METHOD PRIVATE FlagOpenEntity : BOOL
VAR_INPUT
	Identifier : STRING(255);	
END_VAR
VAR_IN_OUT
	Header : CuHeader;
END_VAR
Header.Operator := _operatorInfo.UserName;
Header.OperationsStarted := Context.RealTimeClock.NowLocal();
THIS^.ProcessDataManager.Data.EntityHeader.Results.Result := TcoInspectors.eOverallResult.InProgress;
THIS^.ProcessDataManager.Data._EntityId := Identifier;
THIS^.ProcessDataManager.Data.EntityHeader.OpenOn := THIS^.CuId;
THIS^.ProcessDataManager.Data.EntityHeader.WasReset := FALSE;
END_METHOD

METHOD PRIVATE FlagThrowAwayEntity : BOOL
VAR_IN_OUT	
	CuHeader : CuHeader; 
END_VAR
IF(THIS^.ProcessDataManager.Data.EntityHeader.OpenOn <> eStations.NONE) THEN
	THIS^.ProcessDataManager.Data.EntityHeader.LastStation := THIS^.CuId;
	THIS^.ProcessDataManager.Data.EntityHeader.NextStation := CuHeader.NextOnFailed;
	THIS^.ProcessDataManager.Data.EntityHeader.Results.Result := TcoInspectors.eOverallResult.Failed;
	THIS^.ProcessDataManager.Data.EntityHeader.WasReset := TRUE;
END_IF;
END_METHOD

(*~
	<docu>
		<summary>
			Controls `ground` mode of `CU00x`.
		</summary>
	</docu>
~*)
METHOD Ground : BOOL
VAR_INPUT
END_VAR
(*
	Enable condition to start `groundTask`.
	Modify according your needs.
	[! 
	THIS IS NOT SAFETY CONDITION. THE SAFETY OF PRESONNEL AND EQUIPMENT MUST BE ENSURED BY ADDITIONAL MEANS 
	TO COMPLY WITH REGULATIONS
	]
*)

GroundTask.Task.Enabled :=  THIS^.Technology.AllowGround(inCuId:=CuId)  OR GroundTask.Task.Busy ;

(*
	Invokes `groundTask` from technology object.
*)


IF(Technology.GroundAllTask.Execute()) THEN GroundTask.Restore();GroundTask.Task.Invoke(); END_IF;


IF GroundTask.GroundDone AND GroundTask.Task.Execute() THEN GroundTask.Restore();GroundTask.Task.Invoke();END_IF;
END_METHOD

PROPERTY ABSTRACT GroundTask : REFERENCE TO CUBaseGround
GET
END_GET
END_PROPERTY

PROPERTY FINAL GroupInspection : REFERENCE TO TcoInspectionGroup
GET
GroupInspection REF= _groupInspection;
END_GET
END_PROPERTY

(*~
	<docu>
		<summary>
			Code to be called cylically when `CU00x` idle; no other mode is active.
		</summary>
	</docu>
~*)
METHOD Idle : BOOL
END_METHOD

METHOD InternalCloseEntity : BOOL
VAR_INPUT
	inCarrier : UINT;
	refStorage : REFERENCE TO InternalStorage;
END_VAR
VAR_IN_OUT
	inoHeader : CuHeader; 
END_VAR
VAR_INST
	_internalData : REFERENCE TO InternalStorage;	
END_VAR
THIS^.FlagCloseEntity(inoHeader);
_internalData REF= refStorage;
InternalCloseEntity := _internalData.SaveByCarrier(inCarrier, THIS^.ProcessDataManager.Data);
END_METHOD

METHOD InternalCreateNewEntity : BOOL
VAR_INPUT
	inCarrier : UINT;
	refStorage : REFERENCE TO InternalStorage;
END_VAR
VAR_IN_OUT
	inoHeader : CuHeader; 
END_VAR
VAR_INST
	_internalData : REFERENCE TO InternalStorage;	
END_VAR
THIS^.FlagCreateNewEntity(UINT_TO_STRING(inCarrier), inoHeader);
THIS^.ProcessDataManager.Data.EntityHeader.Carrier := UINT_TO_STRING(inCarrier);
_internalData REF= refStorage;
InternalCreateNewEntity := _internalData.SaveByCarrier(inCarrier, THIS^.ProcessDataManager.Data);
END_METHOD

METHOD InternalFinishEntity : BOOL
VAR_INPUT
	inCarrier : UINT;
	refStorage : REFERENCE TO InternalStorage;
END_VAR
VAR_IN_OUT
	inoHeader : CuHeader; 
END_VAR
VAR_INST
	_internalData : REFERENCE TO InternalStorage;	
END_VAR
THIS^.FlagFinishEntity(inoHeader);

_internalData REF= refStorage;
InternalFinishEntity := _internalData.SaveByCarrier(inCarrier, THIS^.ProcessDataManager.Data);
END_METHOD

METHOD InternalOpenEntity : BOOL
VAR_INPUT
	inCarrier : UINT;
	refStorage : REFERENCE TO InternalStorage;
END_VAR
VAR_IN_OUT
	inoHeader : CuHeader; 
END_VAR
VAR_INST
	_internalData : REFERENCE TO InternalStorage;	
END_VAR
_internalData REF= refStorage;
InternalOpenEntity := _internalData.GetByCarrier(inCarrier, THIS^.ProcessDataManager.Data);
THIS^.FlagOpenEntity(UINT_TO_STRING(inCarrier), inoHeader);
END_METHOD

METHOD InternalRetrieveEntity : BOOL
VAR_INPUT
	inCarrier : UINT;
	refStorage : REFERENCE TO InternalStorage;
END_VAR
VAR_INST
	_internalData : REFERENCE TO InternalStorage;	
END_VAR
_internalData REF= refStorage;
InternalRetrieveEntity := _internalData.GetByCarrier(inCarrier, THIS^.ProcessDataManager.Data);
END_METHOD

METHOD InternalThrowAwayEntity : BOOL
VAR_INPUT
	inCarrier : UINT;
	refStorage : REFERENCE TO InternalStorage;
END_VAR
VAR_IN_OUT
	inoHeader : CuHeader; 
END_VAR
VAR_INST
	_internalData : REFERENCE TO InternalStorage;	
END_VAR
THIS^.FlagThrowAwayEntity(inoHeader);
_internalData REF= refStorage;
InternalThrowAwayEntity := _internalData.SaveByCarrier(inCarrier, THIS^.ProcessDataManager.Data);
END_METHOD

(*~
	<docu>
		<summary>
			Controls `manual` mode of `CU00x`.
		</summary>
	</docu>
~*)
METHOD Manual : BOOL
VAR_INPUT
END_VAR
(*
	Enable condition to start `automatTask`.
	Modify according your needs.
	[! 
	THIS IS NOT SAFETY CONDITION. THE SAFETY OF PRESONNEL AND EQUIPMENT MUST BE ENSURED BY ADDITIONAL MEANS 
	TO COMPLY WITH REGULATIONS
	]
*)

ManualTask.Task.Enabled :=  THIS^.Technology.AllowManual(inCuId:=CuId)  OR ManualTask.Task.Busy;
END_METHOD

PROPERTY ABSTRACT ManualTask : REFERENCE TO TcoTaskedService
GET
END_GET
END_PROPERTY

PROPERTY FINAL ProcessDataManager : REFERENCE TO ProcessDataManager
GET
ProcessDataManager REF= _processData;
END_GET
END_PROPERTY

PROPERTY  ReadEntityTask : TcoCore.ITcoTaskStatus
GET
ReadEntityTask := _processData._readTask;
END_GET
END_PROPERTY

METHOD ReadyForOperations : BOOL
VAR_INPUT
END_VAR
ReadyForOperations := _readyForOperations;
END_METHOD

PROPERTY ABSTRACT RecoverTask : REFERENCE TO CUBaseRecover
GET
END_GET
END_PROPERTY

PROPERTY RecurringFails : REFERENCE TO CuBaseRecurringFailures
GET
RecurringFails REF= _recurringFails;
END_GET
END_PROPERTY

METHOD ResetReadyForOperations : BOOL
_readyForOperations := false;
END_METHOD

METHOD  RunOperations : BOOL
VAR_INPUT
	refGlobalTrigger:REFERENCE TO BOOL;
END_VAR
VAR
	_trrigger:REFERENCE TO BOOL;
END_VAR
_trrigger REF=refGlobalTrigger;
RunOperations := _trrigger;
END_METHOD

METHOD  SetReadyForOperations : BOOL
VAR_INPUT
END_VAR
_readyForOperations := TRUE;
END_METHOD

PROPERTY ABSTRACT StatusInfo : REFERENCE TO CUBaseStatusInfo
GET
END_GET
END_PROPERTY

PROPERTY ABSTRACT SuspendTask : REFERENCE TO CUBaseSuspend
GET
END_GET
END_PROPERTY

PROPERTY Technology : REFERENCE TO Technology
GET
VAR
    _technology : POINTER TO Technology;
END_VAR
IF __QUERYPOINTER(Parent, _technology) THEN // Check if _Parent is Station001
    Technology REF= _technology^;              // If the check is successful dereference a pointer. simlar to THIS^ or SUPER^
END_IF
END_GET
END_PROPERTY

PROPERTY PUBLIC ToggleBlinker : REFERENCE TO TcoUtilities.TcoBlinker
GET
ToggleBlinker ref= _toggle;
END_GET
END_PROPERTY

PROPERTY  UpdateEntityTask : TcoCore.ITcoTaskStatus
GET
UpdateEntityTask := _processData._updateTask;
END_GET
END_PROPERTY

METHOD UpdateInfo : BOOL
VAR_INPUT
END_VAR
_toggle(inOffTime:=T#500MS,inOnTime:=T#500MS);

IF AutomatTask.ClearCounterDataTask.Execute() THEN
	AutomatTask.ClearCounter();
	AutomatTask.ClearCounterDataTask.DoneWhen(TRUE);
END_IF

_statusInfo.State := eCUState.None;

IF _statusInfo.CurrentCleanCycleTime  >= _settings.WarningCycleTime
	AND _statusInfo.CurrentCleanCycleTime  < _settings.ErrorCycleTime THEN
	_statusInfo.State:= eCUState.HasWarning;
ELSIF _statusInfo.CurrentCleanCycleTime   >= _settings.ErrorCycleTime THEN
	_statusInfo.State := eCUState.HasError;
END_IF; 


IF _toggle.IsOff THEN
	_statusInfo.State := eCUState.None;
END_IF



IF AutomatTask.Task.Busy THEN

    _statusInfo.Mode                   := eCUMode.AutomatMode;
    _statusInfo.CurrentTaskDescription := '<#AUTOMAT#>';
    _statusInfo.CurrentCycleTime       := AutomatTask._SequenceElapsedTime;
	_statusInfo.CurrentCleanCycleTime  := T#0S;

	IF AutomatTask._startCleanCycleTime<>T#0S AND AutomatTask._stopCleanCycleTime=T#0S  THEN
		_statusInfo.CurrentCleanCycleTime  := AutomatTask._SequenceElapsedTime-AutomatTask._startCleanCycleTime;
	ELSIF AutomatTask._stopCleanCycleTime<>T#0S  THEN
		_statusInfo.CurrentCleanCycleTime  := AutomatTask._stopCleanCycleTime-AutomatTask._startCleanCycleTime;
	ELSE
		_statusInfo.CurrentCleanCycleTime :=AutomatTask._startCleanCycleTime;
	END_IF;
	
	_statusInfo.AverageCycleTime	   := AutomatTask.AverageCycleTime;
	_statusInfo.AverageCleanCycleTime  := AutomatTask.AverageCleanCycleTime;
    _statusInfo.CurrentUid             := AutomatTask.CurrentStep.ID;
    _statusInfo.CurrentOperation       := AutomatTask.CurrentStep.Description;
    _statusInfo.CurrentIsInStepMode    := AutomatTask._modeController._mode = eSequencerMode.StepMode;
ELSIF GroundTask.Task.Busy THEN
    _statusInfo.Mode := eCUMode.GroundMode;
	_statusInfo.CurrentTaskDescription := '<#GROUND#>';
    _statusInfo.CurrentCycleTime       := GroundTask._SequenceElapsedTime;
	_statusInfo.CurrentCleanCycleTime := T#0S;
	_statusInfo.AverageCycleTime	   := GroundTask.AverageCycleTime;
	_statusInfo.AverageCleanCycleTime  := T#0S;
    _statusInfo.CurrentUid             := GroundTask.CurrentStep.ID;
    _statusInfo.CurrentOperation       := GroundTask.CurrentStep.Description;
    _statusInfo.CurrentIsInStepMode    := GroundTask._modeController._mode = eSequencerMode.StepMode;
ELSIF THIS^.ManualTask.Busy THEN
    _statusInfo.Mode := eCUMode.ManualMode;
	_statusInfo.CurrentTaskDescription := '<#MANUAL#>';
	_statusInfo.State := eCUState.None;
	_statusInfo.CurrentIsInStepMode    := FALSE;

ELSIF THIS^.GroundTask.Task.Done THEN
	_statusInfo.CurrentTaskDescription := '<#READY TO START#>';
	_statusInfo.Mode := eCUMode.GroundModeDone;
	_statusInfo.CurrentCycleTime       := GroundTask._SequenceElapsedTime;
    _statusInfo.CurrentUid             := GroundTask.CurrentStep.ID;
    _statusInfo.CurrentOperation       := GroundTask.CurrentStep.Description;
    _statusInfo.CurrentIsInStepMode    := GroundTask._modeController._mode = eSequencerMode.StepMode;
	_statusInfo.State := eCUState.None;

ELSE
    _statusInfo.Mode := eCUMode.NoMode;	
	_statusInfo.CurrentTaskDescription := '<#IDLE#>';
	_statusInfo.CurrentCycleTime       := T#0S;
    _statusInfo.CurrentUid             := 0;
    _statusInfo.CurrentOperation       := '';
    _statusInfo.CurrentIsInStepMode    := FALSE;
	_statusInfo.State := eCUState.None;
END_IF
END_METHOD

END_FUNCTION_BLOCK

// ---- Technology/Data/ProcessDataManager.TcPOU
FUNCTION_BLOCK ProcessDataManager EXTENDS TcoData.TcoDataExchange
VAR
    _data : ProcessData := (Parent := THIS^);
	_sb : TcoCore.StringBuilder;
END_VAR

SUPER^();

PROPERTY Data : REFERENCE TO ProcessData
GET
Data REF= _data;
END_GET
END_PROPERTY

END_FUNCTION_BLOCK

// ---- Abstractions/CUBase/RemoteTasks/ProductionPlaner.TcPOU
FUNCTION_BLOCK PUBLIC ProductionPlaner EXTENDS TcoCore.TcoRemoteTask
VAR_INPUT
END_VAR
VAR_OUTPUT
END_VAR
VAR
	_productonPlanCompleted: BOOL;
	_productionPlanIsEmpty: BOOL;
	_requiredProcessSettings: STRING;
END_VAR

super^();

PROPERTY PUBLIC ProductionPlanCompleted : bool
GET
ProductionPlanCompleted:=_productonPlanCompleted;
END_GET
END_PROPERTY

PROPERTY PUBLIC ProductionPlanIsEmpty : bool
GET
ProductionPlanIsEmpty:=_productionPlanIsEmpty;
END_GET
END_PROPERTY

PROPERTY RequiredProcessSettingsId : string
GET
RequiredProcessSettingsId:=_requiredProcessSettings;
END_GET
END_PROPERTY

(*~
	<docu>
		<summary>
			Restores this instance to the Ready state. Can be called explicitly or from within one of the restore mechanisms.
			<para>
				See also <see cref="PlcDocu.TcoCore.TcoTask.AutoRestorable()"/>
			</para>
		</summary>			
	</docu>	
~*)
METHOD Restore : ITcoRestorable
SUPER^.Restore();
_productonPlanCompleted:=FALSE;
_productionPlanIsEmpty:=FALSE;
_requiredProcessSettings:='';
END_METHOD

END_FUNCTION_BLOCK

// ---- Technology/Data/InternalStorage.TcPOU
FUNCTION_BLOCK InternalStorage EXTENDS TcoCore.TcoObject 
VAR
	_data : ARRAY[0..40] OF ProcessData; 
END_VAR
VAR CONSTANT
	_maxNumberOfCarriers : UINT := 40;
END_VAR

METHOD GetByCarrier : BOOL
VAR_INPUT
	inCarrier : UINT;
END_VAR
VAR_IN_OUT
	inoData : ProcessData;
END_VAR
IF(inCarrier >= 0 AND inCarrier < _maxNumberOfCarriers) THEN
	inoData := _data[inCarrier];
	GetByCarrier := TRUE;
	RETURN;	
END_IF

Messenger.Post(CONCAT('<#Requested carrier is out of range of internal storage. Max number of carriers is#> ', UINT_TO_STRING(_maxNumberOfCarriers)), eMessageCategory.ProgrammingError);
END_METHOD

METHOD SaveByCarrier : BOOL
VAR_INPUT
	inCarrier : UINT;
END_VAR
VAR_IN_OUT
	inoData : ProcessData;
END_VAR
IF(inCarrier >= 0 AND inCarrier < _maxNumberOfCarriers) THEN
	_data[inCarrier] := inoData;
	SaveByCarrier := TRUE;
	RETURN;	
END_IF

Messenger.Post(CONCAT('<#Requested carrier is out of range of internal storage. Max number of carriers is#> ', UINT_TO_STRING(_maxNumberOfCarriers)), eMessageCategory.ProgrammingError);
END_METHOD

END_FUNCTION_BLOCK

// ---- Technology/Technology.TcPOU
FUNCTION_BLOCK Technology EXTENDS TcoCore.TcoContext
VAR	
    _processSettings     : ProcessDataManager(THIS^);  			//a.k.a receipe
	_reworkSettings     : ProcessDataManager(THIS^);  			//a.k.a receipe for rework
    _technologySettings  : TechnologicalDataManager(THIS^);		//a.k.a machine settings
    _processTraceability : ProcessDataManager(THIS^);			//the same structure as process setting but filled with actual production data (measurements, inspection results, etc)
	_internalStorage : InternalStorage(THIS^);					//

	
	fbGetCurTaskIndex            : GETCURTASKINDEX;
	_notificationPanel      : NotificationPanel(THIS^);				//provide technology state signals to side baner in visualisation
    {attribute addProperty Name "<#AUTOMAT ALL#>"}
    _automatAllTask : TcoCore.TcoTask(THIS^);					// Commmand-like taks to execute automation mode on whole technology. Handled in controlled units.
    {attribute addProperty Name "<#GROUND ALL#>"}
    _groundAllTask : TcoCore.TcoTask(THIS^);	

	{attribute addProperty Name "<#_cu00x#>"}					
    _cu00x         : CU00x(THIS^);
	
	{attribute addProperty Name "<#Technology Components#>"}	
	_components : TechnologyComponents:= (Parent := THIS^);

	{attribute addProperty Name "Device 1 (EtherCAT)"}
	Device_1 : TcoIo.TcoEthercatMasterDevice(THIS^);
	
	_setDummyConditionsSuffisient:BOOL;
	_dummyBlinker              : TcoUtilities.TcoBlinker(THIS^);
	_runOperations:BOOL;

	
END_VAR

METHOD AllowAutomat : BOOL
VAR_INPUT
	inCuId : eStations;
END_VAR

VAR
	retVal: BOOL;
END_VAR
retVal := FALSE;
IF inCuId = eStations.CU00x THEN
	 retVal := TRUE;// Components.Zone1.Status.State.AnyKeyManual AND Components.ControlVoltages.R1.GlobalControlVoltage.Signal;
END_IF;


AllowAutomat := retVal;
END_METHOD

METHOD AllowGround : BOOL
VAR_INPUT
	inCuId : eStations;
END_VAR

VAR
	retVal: BOOL;
END_VAR
retVal := FALSE;
IF inCuId = eStations.CU00x THEN
	 retVal := TRUE;// Components.Zone1.Status.State.AnyKeyManual AND Components.ControlVoltages.R1.GlobalControlVoltage.Signal;
END_IF;


AllowGround := retVal;
END_METHOD

METHOD AllowManual :  BOOL
VAR_INPUT
	inCuId : eStations;
END_VAR


VAR
	retVal: BOOL;
END_VAR
retVal := FALSE;
IF inCuId = eStations.CU00x THEN
	 retVal := TRUE;// Components.Zone1.Status.State.AnyKeyManual AND Components.ControlVoltages.R1.GlobalControlVoltage.Signal;
END_IF;


AllowManual := retVal;
END_METHOD

PROPERTY AutomatAllTask : REFERENCE TO TcoCore.TcoTask
GET
AutomatAllTask REF= _automatAllTask;
END_GET
END_PROPERTY

PROPERTY Components : REFERENCE TO TechnologyComponents
GET
Components REF= _components;
END_GET
END_PROPERTY

PROPERTY PUBLIC Cu00x : Reference to CU00x
GET
Cu00x REF=_cu00x;
END_GET
END_PROPERTY

METHOD ForceStepMode : BOOL
ForceStepMode := FALSE;
END_METHOD

PROPERTY GroundAllTask : REFERENCE TO TcoCore.TcoTask
GET
GroundAllTask REF= _groundAllTask;
END_GET
END_PROPERTY

METHOD InitializeComponents
VAR_INPUT
END_VAR

VAR
	controlVolage: BOOL;
	controlVoltageDoor: BOOL;
	estop: BOOL;
	presure: BOOL;
	locked: BOOL;
	lock: BOOL;
	opened: BOOL;
	closed: BOOL;
	
END_VAR
controlVolage:=FALSE;
controlVoltageDoor:=FALSE;
estop:=FALSE;
presure:=FALSE;

//_dummyBlinker(inOffTime := T#10000MS, inOnTime := T#10000MS);
(*
closed:=GVL_iXlinker.EC1.EK1200.IA1_EL1809.Channel_8.Input;
locked:=GVL_iXlinker.EC1.EK1200.IA1_EL1809.Channel_9.Input;

IF _setDummyConditionsSuffisient THEN
	controlVolage:=TRUE;
	controlVoltageDoor:=TRUE;
	estop:=FALSE;
	presure:=TRUE;


END_IF;

_components.ModeKey(inoKeyState1:=GVL_iXlinker.EC1.EK1200.IA1_EL1809.Channel_1.Input ,
					inoKeyState2:=GVL_iXlinker.EC1.EK1200.IA1_EL1809.Channel_2.Input);
					
_components.NormalServiceKey(inoSignal:=GVL_iXlinker.EC1.EK1200.IA1_EL1809.Channel_3.Input);
					
_components.ControlButtons(
	inoButtonRecover:=GVL_iXlinker.EC1.EK1200.IA1_EL1809.Channel_4.Input  , 
	inoButtonSuspend:=GVL_iXlinker.EC1.EK1200.IA1_EL1809.Channel_5.Input  , 
	inoButtonGround:=GVL_iXlinker.EC1.EK1200.IA1_EL1809.Channel_6.Input , 
	inoButtonAuto:=GVL_iXlinker.EC1.EK1200.IA1_EL1809.Channel_7.Input, 
	inoButtonRecoverLight:=GVL_iXlinker.EC1.EK1200.QA1_EL2809.Channel_1.Output  , 
	inoButtonSuspendLight:=GVL_iXlinker.EC1.EK1200.QA1_EL2809.Channel_2.Output  , 
	inoButtonGroundLight:=GVL_iXlinker.EC1.EK1200.QA1_EL2809.Channel_3.Output  , 
	inoButtonAutoLight:= GVL_iXlinker.EC1.EK1200.QA1_EL2809.Channel_4.Output );
	

					

_components.GlobalControlVoltage(inoSignal := controlVolage);

_components.LocalControlVoltage(inoSignal := controlVolage);
_components.LocalDoorVoltage(inoSignal := controlVoltageDoor);

_components.EmergencyStop(inoSignal := estop);
_components.AirPresureOk(inoSignal:= presure);


_components.StandardDoor(inoIsLocked := locked,
    inoIsOpen := opened,
    inoLock :=lock);
	
	
_components.BasicDoor(inoIsClosed := closed,
     inoLock := lock);


_components.DoorCicuit();

_components.Zone(inDoorCircuit:=_components.DoorCicuit,
				inEstopActive:=_components.EmergencyStop.Signal,
				inAirPressureOK:= _components.AirPresureOk.Signal);
		
				
_components.Zone.Service();
*)
END_METHOD

METHOD InitializeComponentsOnce
VAR_INPUT
END_VAR
_components.DoorCicuit.Restore();
_components.Zone.Restore();



_components.DoorCicuit.AddDoors(inDoor:=_components.StandardDoor);
_components.DoorCicuit.AddDoors(inDoor:=_components.BasicDoor);
_components.DoorCicuit.AddGlobalVoltage(inVoltage:=_components.GlobalControlVoltage);
_components.DoorCicuit.AddLocalVoltage(inVoltage:=_components.LocalControlVoltage);
_components.DoorCicuit.AddLocalDoorsVoltage(inVoltage:=_components.LocalDoorVoltage);


_components.Zone.AddControlledUnit(inControlledUnit:=_cu00x);
_components.Zone.AddControlButtons(inControlButtons:=_components.ControlButtons);
_components.Zone.AddKeyMode(inKeyMode:=_components.ModeKey);
_components.Zone.AddKeyNormalService(inKeyNormalService:=_components.NormalServiceKey);
END_METHOD

PROPERTY InternalStorage : REFERENCE TO InternalStorage
GET
InternalStorage REF= _internalStorage;
END_GET
END_PROPERTY

(*~
	<docu>
		<summary>
			Main method of the TcoContext. This is the entry point of any control logic that belongs to this context. 
			The call of this method is ensured by calling the <c>InstanceName.Run()</c> method, and it must not be called explicitly.
			This method is abstract, and it must be overridden in derived block.
		</summary>
	</docu>
~*)
METHOD PROTECTED Main
VAR
	_notificationSourceSignals: NotificationPanelInfo;
	safetyCircuitOk: BOOL;
	_eStopActive: BOOL;
	_keysAto: BOOL;
	_closed: BOOL;
	_locked: BOOL;
END_VAR
(*
	Context settings 
*)

// RTC Synchronisation
THIS^.RtcSynchronize(TRUE,  
					 '192.168.4.1.1.1',    // Provide AMS ID of the time source, leave blank if local. 
					 60);

// Messenger logger settings
_settings.Messaging.MessageDigestMethod := eMessageDigestMethod.CRC32;
_settings.Messaging.MessengerLoggingMethod := eMessengerLogMethod.OnEventRisen;


_components.DoorCicuit.Config.MaxDoors:=12;
_components.DoorCicuit.Config.MaxGlobalVoltage:=2;
_components.DoorCicuit.Config.MaxLocalVoltage:=2;
_components.DoorCicuit.Config.MaxLocalDoorsVoltage:=2;


_components.Zone.Config.MaxControlButtons:=2;
_components.Zone.Config.MaxControledUnits:=10;
_components.Zone.Config.MaxKeyMode:=2;
_components.Zone.Config.MaxKeyNormalService:=2;



THIS^.InitializeComponents();
fbGetCurTaskIndex();
IF _TaskInfo[fbGetCurTaskIndex.index].FirstCycle THEN
    // The code that you want to be executed at the first cycle of  PLC only 
	THIS^.InitializeComponentsOnce();
END_IF

//notification panel
 Context.Environment.Messaging.Suspend();
			
_closed:=TRUE;
//_closed   := 	Components.Safety.DoorCircuits.DoorCircuit_2.IsClosed 
//			AND Components.Safety.DoorCircuits.DoorCircuit_3.IsClosed  
//			AND Components.Safety.DoorCircuits.DoorCircuit_4.IsClosed  
//			AND Components.Safety.DoorCircuits.DoorCircuit_5.IsClosed  
//			AND Components.Safety.DoorCircuits.DoorCircuit_6.IsClosed;

 _locked:=TRUE;
//_locked   := 	Components.Safety.DoorCircuits.DoorCircuit_2.IsLocked 
//			AND Components.Safety.DoorCircuits.DoorCircuit_3.IsLocked  
//			AND Components.Safety.DoorCircuits.DoorCircuit_4.IsLocked  
//			AND Components.Safety.DoorCircuits.DoorCircuit_5.IsLocked  
//			AND Components.Safety.DoorCircuits.DoorCircuit_6.IsLocked;
			
_keysAto  := TRUE;
_eStopActive:=0;


_notificationSourceSignals.ControlVoltage   := TRUE;//Components.ControlVoltage.Signal.Signal 
_notificationSourceSignals.AirPressure      := TRUE;//Components.AirPressureOk.Signal.Signal, 
_notificationSourceSignals.AutomatAllowed   := _keysAto; 
_notificationSourceSignals.EmergencyStop    := _eStopActive > 0; 
_notificationSourceSignals.SafetyDoorOk     :=safetyCircuitOk;	
_notificationSourceSignals.LightCurtain     := TRUE; 	// not used
_notificationSourceSignals.DoorClosed       := _closed; 
_notificationSourceSignals.DoorLocked       := _locked; 
_notificationSourceSignals.ProcessDataOk    := _processSettings._data._EntityId <> '';
_notificationSourceSignals.TechnologyDataOk := _technologySettings._data._EntityId <> '';  
	
_notificationPanel(inBlinkPeriod:=T#500MS , inSignalSource:=_notificationSourceSignals );
			
 Context.Environment.Messaging.Resume();

(*
	
	Data managers

*)

_processSettings();
_reworkSettings();
_technologySettings();

(*

	Controlled units
	
*)

_cu00x();


_automatAllTask();
_groundAllTask();

//Device_1(	SyncUnits		:= ADR(		GVL_iXlinker.EC1.SyncUnits),
//			SyncUnitsSize	:= SIZEOF(	GVL_iXlinker.EC1.SyncUnits),
//			Inputs			:=			GVL_iXlinker.EC1.Inputs,
//			InfoData		:=			GVL_iXlinker.EC1.InfoData);
END_METHOD


(*~
	<docu>
		<summary>
			Called upon exit from the context. When overridden in derived class allows to execute an arbitrary logic after closing the context cycle.	
		</summary>			
	</docu>	
~*)METHOD PROTECTED OnExit
_automatAllTask.DoneWhen(TRUE);
_groundAllTask.DoneWhen(TRUE);
END_METHOD

PROPERTY ProcessSettings : REFERENCE TO ProcessDataManager
GET
ProcessSettings REF= _processSettings;
END_GET
END_PROPERTY

PROPERTY ReworkSettings : REFERENCE TO ProcessDataManager
GET
ReworkSettings REF= _reworkSettings;
END_GET
END_PROPERTY

PROPERTY RunOperations : REFERENCE TO BOOL
GET
RunOperations REF= _runOperations;
END_GET
END_PROPERTY

PROPERTY TechnologicalSettings : REFERENCE TO TechnologicalDataManager
GET
TechnologicalSettings REF= _technologySettings;
END_GET
END_PROPERTY

END_FUNCTION_BLOCK

// ---- Abstractions/Generic/NotificationPanel/NotificationPanel.TcPOU
{attribute wpf [Container(Layout.Stack)]}
FUNCTION_BLOCK NotificationPanel EXTENDS TcoObject
VAR_INPUT
	(*~
		<docu>
			<summary>
				Time duration for toggle signal.
			</summary>
		</docu>
	~*)
	inBlinkPeriod:TIME;
END_VAR

VAR
	{attribute addProperty Name "<#Heart beat#>"}
  	_heartBeat : BOOL;
	
    {attribute clr [RenderIgnore()]}
	_badgeValue : INT;

	{attribute clr [RenderIgnore()]}
    _toggle: TcoUtilities.TcoBlinker(THIS^);
	
	_iconSet: ARRAY[0..20] OF Icon; //ak potrebujes zobrazit viac ikon, uprav velkost pola
	
	_iconSetClear : ARRAY[0..20] OF Icon; //ak potrebujes zobrazit viac ikon, uprav velkost pola
	
	_iconPlcPulse : Icon;
	
	_iconParamsClear : Icon;
	
END_VAR



_iconPlcPulse.Title := '<#PLC connection#>';
_iconPlcPulse.IconType := TO_STRING(eIconType.plcConnection);
_iconPlcPulse.Signal := _heartBeat;
_iconPlcPulse.DisableRedIcon := TRUE;
addIcon(_iconPlcPulse);

//setIconsStyle();

Blink();
CountSignals();

METHOD AddIcon : BOOL
VAR_INPUT
	inIcon : Icon;
END_VAR

VAR 
	_index : INT;
END_VAR
FOR  _index := 0 TO 20 DO 
	IF _IconSet[_index].Title = '' THEN
		_IconSet[_index] := inIcon;
		RETURN;
	END_IF
END_FOR
END_METHOD

METHOD Blink
VAR 
	_index : INT;
END_VAR
_toggle(inOffTime:=inBlinkPeriod,inOnTime:=inBlinkPeriod);
_heartBeat := _toggle.IsOn;
	FOR _index := 0 TO 20 DO
		IF _iconSet[_index].BlinkEnabled AND NOT _iconSet[_index].Signal THEN 
			_iconSet[_index].SignalBlink := _toggle.IsOn;		
		ELSE
			_iconSet[_index].SignalBlink := _iconSet[_index].Signal;
		END_IF
	END_FOR
END_METHOD

METHOD Clear
_iconSet := _iconSetClear;
_badgeValue := 0;
END_METHOD

METHOD CountSignals
VAR
	_iconIndex : INT;
END_VAR
_iconIndex := 0;
_badgeValue := 0;
FOR _iconIndex := 0 TO 20 DO
	IF _iconSet[_iconIndex].Title <> '' AND  NOT _iconSet[_iconIndex].DisableRedIcon THEN 
		_badgeValue := _badgeValue + BOOL_TO_INT(NOT _iconSet[_iconIndex].Signal);
	END_IF
END_FOR
END_METHOD

METHOD PRIVATE setIconsStyle
VAR 
	_index : INT;
END_VAR
//FOR _index := 0 TO 20 DO 
//	CASE _iconSet[_index].IconType OF 
//		eIconType.controlVoltage : _iconSet[_index].IconType := 'Power';
//		eIconType.airPressure : _iconSet[_index].IconType := 'OxygenTank';
//		eIconType.emergencyStop : _iconSet[_index].IconType := 'Alert';
//		eIconType.safetyDoor : _iconSet[_index].IconType := 'ShieldCheck';
//		eIconType.doorClosed : _iconSet[_index].IconType := 'Door';
//		eIconType.doorLocked : _iconSet[_index].IconType := 'DoorClosedLock';
//		eIconType.processDataLoaded : _iconSet[_index].IconType := 'CogOutline';
//		eIconType.technologyDataLoaded : _iconSet[_index].IconType := 'ClipboardCheckOutline';
//		eIconType.opticBarrier : _iconSet[_index].IconType := 'Hand';
//		eIconType.robot : _iconSet[_index].IconType := 'RobotIndustrial';
//		eIconType.plcConnection : _iconSet[_index].IconType := 'HeartPulse';
//	ELSE
//		 _iconSet[_index].IconType := _iconSet[_index].IconType;
//	END_CASE
//END_FOR
END_METHOD

METHOD SetSignal
VAR_INPUT
	inTitle : STRING;
	inSignal : BOOL;
END_VAR

VAR
	_index : INT;
END_VAR
FOR _index := 0 TO 20 DO 
	IF _iconSet[_index].Title = inTitle THEN 
		_iconSet[_index].Signal := inSignal;
		RETURN;
	END_IF
END_FOR
END_METHOD

END_FUNCTION_BLOCK

// ---- Technology/CU00x/CU00x.TcPOU
{attribute addProperty ShortName "CU00x"}
{attribute addProperty Name "Controlled unit x_tempalte_x"}
FUNCTION_BLOCK CU00x EXTENDS CUBase 
VAR
    _cuProcessDataDisplay       :  CU00xProcessData := (Parent := THIS^);
    _cuTechnologicalDataDisplay :  CU00xTechnologicalData := (Parent := THIS^);
    _components          		:  CU00xComponents := (Parent := THIS^);
	{attribute addProperty Name "<#MANUAL#>"}
    {attribute addProperty ToolTip "<#Start manual/Service mode#>"}	
    _manualTask : CU00xManualTask(THIS^);
	{attribute addProperty Name "<#GROUND#>"}
	{attribute addProperty ToolTip "<#Brings the device into basic position.#>"}
	_groundTask : CU00xGroundTask(THIS^, TcoCore.eRestoreMode.None);
	{attribute addProperty Name "<#AUTOMAT#>"}
	{attribute addProperty ToolTip "<#Starts automatic sequence. Before start you need to perform grounding sequence.#>"}	
	_automatTask : CU00xAutomatTask(THIS^, TcoCore.eRestoreMode.None);     
	{attribute addProperty Name "<#SUSPEND PROCESS#>"}
    {attribute addProperty ToolTip "<#Starts suspend sequence of process(automatic,ground sequence).#>"}	
    _suspendTask : CU00xSuspendTask(THIS^, TcoCore.eRestoreMode.None);     
	{attribute addProperty Name "<#RECOVER PROCESS#>"}
    {attribute addProperty ToolTip "<#Starts suspend sequence of process(automatic,ground sequence).#>"}	
    _recoverTask : CU00xRecoverTask(THIS^, TcoCore.eRestoreMode.None);     
  	
	{attribute addProperty Name "<#Test positions#>"}
	_positions : Cu00xTestPositions(THIS^);

	{attribute addProperty Name "<#Test multi positions#>"}
	_positionsMulti : CU00xTestMultiPositions(THIS^);
	

END_VAR

THIS^.CuId := eStations.CU00x;



(*
	This controlled unit's component initialization.
*)

THIS^.InitializeComponents();

(*
	This controlled unit process data crud operations handler.
	Control exchange of process data between this controlled unit and the data repository.
*)

_processData();
_productionPlaner();


(*
	
	Cu's Modes
	
*)

Automat();
Ground();
Manual();


_suspendTask();
_recoverTask();







(*
	When no mode is active 'Idle' method should be called.
	'NoMode' method shouls contain code that renders this cu idle. 
*)

IF NOT (AutomatTask.Task.Busy 
		OR GroundTask.Task.Busy
		OR ManualTask.Task.Busy) 
THEN
	Idle();
END_IF



(*
	Updates this controlled unit's information for the UI.
*)


UpdateInfo();

_cuProcessDataDisplay := ProcessDataManager.Data.CU00x;
_cuTechnologicalDataDisplay := Technology.TechnologicalSettings.Data.CU00x;

_settings.WarningCycleTime:= _cuTechnologicalDataDisplay.WarningCycleTime;
_settings.ErrorCycleTime:= _cuTechnologicalDataDisplay.ErrorCycleTime;
_settings.AnyRecurringFailure:= _cuTechnologicalDataDisplay.AnyRecurringFailure;
_settings.SameRecurringFailure:= _cuTechnologicalDataDisplay.SameRecurringFailure;

(*~
	<docu>
		<summary>
			Controls `automatic` mode of `CU00x`.
		</summary>
	</docu>
~*)
METHOD Automat
VAR_INPUT
END_VAR
(*
	Enable condition to start `automatTask`.
	Modify according your needs.
	[! 
	THIS IS NOT SAFETY CONDITION. THE SAFETY OF PRESONNEL AND EQUIPMENT MUST BE ENSURED BY ADDITIONAL MEANS 
	TO COMPLY WITH REGULATIONS
	]
*)


//_automatTask.Task.Enabled := (_groundTask.GroundDone OR  _automatTask.Task.Busy) AND THIS^.Technology.AllowAutomat();

(*
	Invokes `groundTask` from technology object.
*)

//IF(Technology.AutomatAllTask.Execute()) THEN _automatTask.Task.Invoke(); END_IF;

//IF(Technology.ForceStepMode()) THEN
 //	_automatTask.ModeController.Mode := eSequencerMode.StepMode;
//END_IF 



(*
	or use default behavior from abstraction
*)
	SUPER^.Automat();

(*

	Executes sequence of automatic mode.

*)

_automatTask();
END_METHOD

PROPERTY AutomatTask : REFERENCE TO CUBaseAutomat
GET
AutomatTask REF= _automatTask;
END_GET
END_PROPERTY

PROPERTY Components : REFERENCE TO CU00xComponents
GET
Components REF= _components;
END_GET
END_PROPERTY

PROPERTY CuProcessData : REFERENCE TO CU00xProcessData
GET
CuProcessData ref=ProcessDataManager.Data.CU00x;
END_GET
END_PROPERTY

(*~
	<docu>
		<summary>
			Controls `ground` mode of `CU00x`.
		</summary>
	</docu>
~*)
METHOD Ground : BOOL
VAR_INPUT
END_VAR
(*
	Enable condition to start `groundTask`.
	Modify according your needs.
	[! 
	THIS IS NOT SAFETY CONDITION. THE SAFETY OF PRESONNEL AND EQUIPMENT MUST BE ENSURED BY ADDITIONAL MEANS 
	TO COMPLY WITH REGULATIONS
	]
*)

//_groundTask.Task.Enabled :=  THIS^.Technology.AllowGround();

(*
	Invokes `groundTask` from technology object.
*)

//IF(Technology.GroundAllTask.Execute()) THEN _groundTask.Task.Invoke(); END_IF;


//IF _groundTask.GroundDone AND _groundTask.Task.Execute() THEN _groundTask.Restore();_groundTask.Task.Invoke();END_IF;


(*
	or use default behavior from abstraction
*)
	SUPER^.Ground();




(*

	Executes sequence of groundTask.

*)

_groundTask();
END_METHOD

PROPERTY GroundTask : REFERENCE TO CUBaseGround
GET
GroundTask REF= _groundTask;
END_GET
END_PROPERTY

(*~
	<docu>
		<summary>
			Code to be called cylically when `CU00x` idle; no other mode is active.
		</summary>
	</docu>
~*)
METHOD Idle : BOOL
END_METHOD

METHOD InitializeComponents : BOOL

VAR_INST
	tempBoolHome: BOOL;
	tempBoolWork: BOOL;
	tempBoolP4Home: BOOL;
	tempBoolP4Work: BOOL;
END_VAR

Components.PairTagTask();
Components.ReworkInstructionTask();
(*
components.Group1.horizontalCylinder(inoAtHomePos:=GVL_iXlinker.EC1.EK1200.IA1_EL1809.Channel_1.Input, 
							   inoAtWorkPos:=GVL_iXlinker.EC1.EK1200.IA1_EL1809.Channel_2.Input, 
							   inoToHomePos:=GVL_iXlinker.EC1.EK1200.IA1_EL1809.Channel_3.Input, 
							   inoToWorkPos:=GVL_iXlinker.EC1.EK1200.IA1_EL1809.Channel_4.Input);
Components.SingleAxis.Config.InfoTime:=T#4S;
Components.SingleAxis.Config.ErrorTime:=T#10S;



Components.SingleAxis(inEnable := ,
    inEnablePositive := ,
    inEnableNegative := ,
    inCalibrationCam := ,
    refAxis := GVL_iXlinker.Axis1,
	inoPositions:= _positions);
	
	

//Components.PickAndPlace();
//Components.PickAndPlace.Service();
		
Components.MultiAxis(inEnableAxis1 := ,
    inEnablePositiveAxis1 := ,
    inEnableNegativeAxis1 := ,
    inCalibrationCamAxis1 := ,
    refAxis1 := GVL_iXlinker.Axis1,
	inoPositions:= _positionsMulti);
	
			
//Components.PickAndPlace.Components.Manipulator(inEnableAxis1 := ,
//    inEnablePositiveAxis1 := ,
//    inEnableNegativeAxis1 := ,
//    inCalibrationCamAxis1 := ,
//    refAxis1 := GVL_iXlinker.Axis1,
//	inoPositions:= _positionsMulti);
*)

Components.PlsPaletizator.Components.I1_PresentBlisterEntry(inoSignal:=GVL_iXlinker.Ec.EC.EK.AB23.Channel_1.Input);
Components.PlsPaletizator.Components.I2_PresentBlisterEntryEmptySpace(inoSignal:=GVL_iXlinker.Ec.EC.Ek.AB23.Channel_2.Input);
Components.PlsPaletizator.Components.I3_PresentBlistersInBufferEmpty(inoSignal:=GVL_iXlinker.Ec.EC.Ek.AB23.Channel_3.Input);
Components.PlsPaletizator.Components.I4_PresentBlisterInWorkingPos(inoSignal:=GVL_iXlinker.Ec.EC.Ek.AB23.Channel_4.Input);
Components.PlsPaletizator.Components.I5_OutBlistersIsThrowedCorrectly(inoSignal:=GVL_iXlinker.Ec.EC.Ek.AB23.Channel_5.Input);
Components.PlsPaletizator.Components.I6_OutBlistersLisftSignal(inoSignal:=GVL_iXlinker.Ec.EC.Ek.AB23.Channel_6.Input);
Components.PlsPaletizator.Components.I7_OutBlistersIsAboveOutBuffer(inoSignal:=GVL_iXlinker.Ec.EC.Ek.AB23.Channel_7.Input);
Components.PlsPaletizator.Components.I8_OutBlistersBufferIsFull(inoSignal:=GVL_iXlinker.Ec.EC.Ek.AB23.Channel_8.Input);



Components.PlsPaletizator.Components.P1_VerticalSepareEntryBlisters
				(inoAtHomePos:=GVL_iXlinker.Ec.EC.Ek.AB21.Channel_1.Input,
				inoAtWorkPos:=GVL_iXlinker.Ec.EC.Ek.AB21.Channel_2.Input,
				inoToHomePos:=tempBoolHome,
				inoToWorkPos:=tempBoolWork);
GVL_iXlinker.Ec.EC.Ek.PNEU.Modules.Outputs.digital_Data_O[0].1:=tempBoolHome;
GVL_iXlinker.Ec.EC.Ek.PNEU.Modules.Outputs.digital_Data_O[0].0:=tempBoolWork;

Components.PlsPaletizator.Components.P2_VerticalSepareEntryBlisters
				(inoAtHomePos:=GVL_iXlinker.Ec.EC.Ek.AB21.Channel_3.Input,
				inoAtWorkPos:=GVL_iXlinker.Ec.EC.Ek.AB21.Channel_4.Input,
				inoToHomePos:=tempBoolHome,
				inoToWorkPos:=tempBoolWork);
GVL_iXlinker.Ec.EC.Ek.PNEU.Modules.Outputs.digital_Data_O[0].3:=tempBoolHome;
GVL_iXlinker.Ec.EC.Ek.PNEU.Modules.Outputs.digital_Data_O[0].2:=tempBoolWork;


Components.PlsPaletizator.Components.P3_HorizontalSepareEntryBlisters
				(inoAtHomePos1:=GVL_iXlinker.Ec.EC.Ek.AB21.Channel_5.Input,
				inoAtWorkPos1:=GVL_iXlinker.Ec.EC.Ek.AB21.Channel_6.Input,
				inoAtHomePos2:=GVL_iXlinker.Ec.EC.Ek.AB21.Channel_7.Input,
				inoAtWorkPos2:=GVL_iXlinker.Ec.EC.Ek.AB21.Channel_8.Input,
				inoToHomePos:=tempBoolHome,
				inoToWorkPos:=tempBoolWork);
GVL_iXlinker.Ec.EC.Ek.PNEU.Modules.Outputs.digital_Data_O[0].5:=tempBoolHome;
GVL_iXlinker.Ec.EC.Ek.PNEU.Modules.Outputs.digital_Data_O[0].4:=tempBoolWork;

Components.PlsPaletizator.Components.P4_FeedEntryBlister
				(inoAtHomePos:=GVL_iXlinker.Ec.EC.Ek.AB21.Channel_9.Input,
				inoAtWorkPos:=GVL_iXlinker.Ec.EC.Ek.AB21.Channel_10.Input,
				inoToHomePos:=tempBoolP4Home,
				inoToWorkPos:=tempBoolP4Work);
				

GVL_iXlinker.Ec.EC.Ek.PNEU.Modules.Outputs.digital_Data_O[0].7:=tempBoolP4Home;
GVL_iXlinker.Ec.EC.Ek.PNEU.Modules.Outputs.digital_Data_O[0].6:=tempBoolP4Work;

Components.PlsPaletizator.Components.P5_HorizontalSepareOutBlisters
				(inoAtHomePos1:=GVL_iXlinker.Ec.EC.Ek.AB21.Channel_11.Input,
				inoAtWorkPos1:=GVL_iXlinker.Ec.EC.Ek.AB21.Channel_12.Input,
				inoAtHomePos2:=GVL_iXlinker.Ec.EC.Ek.AB21.Channel_13.Input,
				inoAtWorkPos2:=GVL_iXlinker.Ec.EC.Ek.AB21.Channel_14.Input,
				inoToHomePos:=tempBoolHome,
				inoToWorkPos:=tempBoolWork);
GVL_iXlinker.Ec.EC.Ek.PNEU.Modules.Outputs.digital_Data_O[1].1:=tempBoolHome;
GVL_iXlinker.Ec.EC.Ek.PNEU.Modules.Outputs.digital_Data_O[1].0:=tempBoolWork;

Components.PlsPaletizator.Components.P6_VerticalSepareOutBlister
				(inoAtHomePos:=GVL_iXlinker.Ec.EC.Ek.AB21.Channel_15.Input,
				inoAtWorkPos:=GVL_iXlinker.Ec.EC.Ek.AB21.Channel_16.Input,
				inoToHomePos:=tempBoolHome,
				inoToWorkPos:=tempBoolWork);
GVL_iXlinker.Ec.EC.Ek.PNEU.Modules.Outputs.digital_Data_O[1].3:=tempBoolHome;
GVL_iXlinker.Ec.EC.Ek.PNEU.Modules.Outputs.digital_Data_O[1].2:=tempBoolWork;


Components.PlsPaletizator.Components.P7_SupportEntryBlister
				(inoAtHomePos:=GVL_iXlinker.Ec.EC.Ek.AB22.Channel_1.Input,
				inoAtWorkPos:=GVL_iXlinker.Ec.EC.Ek.AB22.Channel_2.Input,
				inoToHomePos:=tempBoolHome,
				inoToWorkPos:=tempBoolWork);
GVL_iXlinker.Ec.EC.Ek.PNEU.Modules.Outputs.digital_Data_O[2].1:=tempBoolHome;
GVL_iXlinker.Ec.EC.Ek.PNEU.Modules.Outputs.digital_Data_O[2].0:=tempBoolWork;

Components.PlsPaletizator.Components.P8_FixEntryBlisterSide
				(inoAtHomePos1:=GVL_iXlinker.Ec.EC.Ek.AB22.Channel_3.Input,
				inoAtWorkPos1:=GVL_iXlinker.Ec.EC.Ek.AB22.Channel_4.Input,
				inoAtHomePos2:=GVL_iXlinker.Ec.EC.Ek.AB22.Channel_5.Input,
				inoAtWorkPos2:=GVL_iXlinker.Ec.EC.Ek.AB22.Channel_6.Input,
				inoToHomePos:=tempBoolHome,
				inoToWorkPos:=tempBoolWork);
GVL_iXlinker.Ec.EC.Ek.PNEU.Modules.Outputs.digital_Data_O[2].3:=tempBoolHome;
GVL_iXlinker.Ec.EC.Ek.PNEU.Modules.Outputs.digital_Data_O[2].2:=tempBoolWork;

Components.PlsPaletizator(inSafeCondition:=GVL_iXlinker.Ec.EC.IA1.Channel_1.Input);
Components.PlsPaletizator.Service();
END_METHOD

(*~
	<docu>
		<summary>
			Controls `manual` mode of `CU00x`.
		</summary>
	</docu>
~*)
METHOD Manual : BOOL
VAR_INPUT
END_VAR
(*
	Enable condition to start `automatTask`.
	Modify according your needs.
	[! 
	THIS IS NOT SAFETY CONDITION. THE SAFETY OF PRESONNEL AND EQUIPMENT MUST BE ENSURED BY ADDITIONAL MEANS 
	TO COMPLY WITH REGULATIONS
	]
*)

	//_manualTask.Task.Enabled := THIS^.Technology.AllowManual();

	
(*
	or use default behavior from abstraction
*)
	SUPER^.Manual();
	

(*

	Executes sequence of manualTask.

*)
_manualTask();
END_METHOD

PROPERTY ManualTask : REFERENCE TO TcoTaskedService
GET
ManualTask REF= _manualTask;
END_GET
END_PROPERTY

PROPERTY ProductionPlanerTask : REFERENCE TO ProductionPlaner
GET
ProductionPlanerTask REF= _productionPlaner;
END_GET
END_PROPERTY

PROPERTY RecoverTask : REFERENCE TO CUBaseRecover
GET
RecoverTask REF= _recoverTask;
END_GET
END_PROPERTY

PROPERTY StatusInfo : REFERENCE TO CUBaseStatusInfo
GET
StatusInfo ref= _statusInfo;
END_GET
END_PROPERTY

PROPERTY SuspendTask : REFERENCE TO CUBaseSuspend
GET
SuspendTask REF= _suspendTask;
END_GET
END_PROPERTY

PROPERTY Technology : REFERENCE TO Technology
GET
VAR
    _technology : POINTER TO Technology;
END_VAR
IF __QUERYPOINTER(Parent, _technology) THEN // Check if _Parent is Station001
    Technology REF= _technology^;              // If the check is successful dereference a pointer. simlar to THIS^ or SUPER^
END_IF
END_GET
END_PROPERTY

PROPERTY TechnologyData : REFERENCE TO CU00xTechnologicalData
GET
TechnologyData ref=_cuTechnologicalDataDisplay;
END_GET
END_PROPERTY

END_FUNCTION_BLOCK

// ---- Technology/CU00x/Manual/CU00xManualTask.TcPOU
FUNCTION_BLOCK CU00xManualTask EXTENDS TcoTaskedService IMPLEMENTS ICUTask
VAR
END_VAR

Run();

(*~
	<docu>
		<summary>
			Main method of the sequener. Custom code needs to be placed here. The sequencer is executed by call of **Instance.Run()** method.
			This method is abstract, and it must be overridden in derived block.
		</summary>
	</docu>
~*)
METHOD PROTECTED Main : BOOL
Messenger.Notify('Running manual mode');
Station.Components.Group1.horizontalCylinder.Service();
Station.Components.Sfk.Service();
END_METHOD

METHOD PROTECTED OnStart
Station.AutomatTask.Restore();
Station.GroundTask.Restore();
Station.GroundTask.CancelGround();
END_METHOD

PROPERTY Station : REFERENCE TO CU00x
GET
VAR
    _station : POINTER TO CU00x;
END_VAR
IF __QUERYPOINTER(Parent, _station) THEN // Check if _Parent is Station001
    Station REF= _station^;              // If the check is successful dereference a pointer. simlar to THIS^ or SUPER^
END_IF
END_GET
END_PROPERTY

END_FUNCTION_BLOCK

// ---- Technology/CU00x/Ground/CU00xGroundTask.TcPOU
FUNCTION_BLOCK CU00xGroundTask EXTENDS CUBaseGround IMPLEMENTS ICUTask

Run();

METHOD DataEntityDiscard
VAR_INPUT	
	inStepID : INT;
	EntityId : STRING(255);
END_VAR
IF (Step(inStepID, TRUE, 'DISCARD ENTITY')) THEN	
    //-------------------------------------		
	IF(Station.ProcessDataManager.Exists(EntityId).Done) THEN
		IF(Station.ProcessDataManager._idExistsTask.Exists) THEN
			StepCompleteWhen(THIS^.Station.EntityFlowDiscard(EntityId, Station.ProcessDataManager.Data.CU00x.Header).Done);
		ELSE
			CompleteStep();
		END_IF
	END_IF;					   		    				
    //-------------------------------------
END_IF
END_METHOD

(*~
	<docu>
		<summary>
			Main method of the sequener. Custom code needs to be placed here. The sequencer is executed by call of **Instance.Run()** method.
			This method is abstract, and it must be overridden in derived block.
		</summary>
	</docu>
~*)
METHOD PROTECTED Main : BOOL
IF (Step(100, TRUE, 'STOPPING OTHER MODES')) THEN
	Station.AutomatTask.ResetCycleTime();//here we can reset averages values of CT
	Station.AutomatTask.Restore();
	Station.ManualTask.Restore();
	Station.ProcessDataManager.Restore();
	Station.AutomatTask.HideAllDialogs();
	Station.GroupInspection.Restore();// hide all dialogs 
    StepCompleteWhen(TRUE);
END_IF

IF (Step(200, TRUE, 'STOPPING OTHER MODES')) THEN	
//	---------------------------------------------------
	
	Station.AutomatTask.ResetCycleTime();
	Station.ProductionPlanerTask.Restore();
	Station.Components.PairTagTask.Restore();
	
	Messenger.Info('INFO MESSAGE');
	
    StepCompleteWhen(THIS^._currentStep.Duration > T#500MS);
//	---------------------------------------------------
END_IF

DataEntityDiscard(5000, THIS^.Station.ProcessDataManager.Data._EntityId);

IF (Step(10000, TRUE, 'LAST STEP')) THEN	
	//---------------------------------------------------
	_groundDone := TRUE;
	THIS^._task.DoneWhen(_groundDone);
	//---------------------------------------------------
END_IF
END_METHOD

METHOD PUBLIC OnStart
SUPER^.OnStart();
Station.AutomatTask.Restore();
Station.ManualTask.Restore();
Station.GroundTask.CancelGround();
END_METHOD

PROPERTY Station : REFERENCE TO CU00x
GET
VAR
    _station : POINTER TO CU00x;
END_VAR
IF __QUERYPOINTER(Parent, _station) THEN // Check if _Parent is Station001
    Station REF= _station^;              // If the check is successful dereference a pointer. simlar to THIS^ or SUPER^
END_IF
END_GET
END_PROPERTY

END_FUNCTION_BLOCK

// ---- Abstractions/Generic/TagsPairing/PairTagTask.TcPOU
FUNCTION_BLOCK PairTagTask EXTENDS TcoCore.TcoRemoteTask
VAR
	
	_key: STRING;
	_assignedValue : STRING;	
	_answerInstruction : STRING(254);
	_answer: TagsPairing;
	{attribute 'hide'}
	_answerClean: TagsPairing;
	_mode: eTagPairingMode;
END_VAR

SUPER^();

PROPERTY Answer : TagsPairing
GET
Answer:=_answer;
END_GET
END_PROPERTY

PROPERTY AnswerInstruction : string
GET
VAR
	retVal: STRING;
END_VAR
AnswerInstruction :=_answerInstruction;
END_GET
END_PROPERTY

(*~
	<docu>
		<summary>
			Restores this instance to the Ready state. Can be called explicitly or from within one of the restore mechanisms.
			<para>
				See also <see cref="PlcDocu.TcoCore.TcoTask.AutoRestorable()"/>
			</para>
		</summary>			
	</docu>	
~*)
METHOD Restore : ITcoRestorable
SUPER^.Restore();
_answer:=_answerClean;
END_METHOD

METHOD Run : REFERENCE TO PairTagTask
VAR_INPUT
	(*~
	<docu>
		<summary>
			The mode is type of operation to be done by invoking  this remote task.(GetTag,CreateTag...)
		</summary>						
	</docu>	
	~*)
	inMode :eTagPairingMode;
	(*~
	<docu>
		<summary>
			The Key is ID  of the tag's Uid on which assigned value will be found . 	
		</summary>						
	</docu>	
	~*)
	inKey : STRING;
		(*~
	<docu>
		<summary>
			The AAssignedValue is user defined additional value, this value provide  better undersanding identification of carriers . 	
		</summary>						
	</docu>	
	~*)
	inAssignedValue : STRING;
	
END_VAR
THIS^._key := inKey;
THIS^._mode := inMode;
THIS^._assignedValue := inAssignedValue;


Run REF= THIS^;
END_METHOD

END_FUNCTION_BLOCK

// ---- Technology/CU00x/Automat/CU00xAutomatTask.TcPOU
FUNCTION_BLOCK CU00xAutomatTask EXTENDS CUBaseAutomat IMPLEMENTS ICUTask
VAR

    _missingProcessSettingMessage : TcoCore.TcoMessenger(THIS^);
    _paralellTask : CU00xAutomatParalell_1_Task(THIS^, TcoCore.eRestoreMode.None);

    _sb : TcoCore.StringBuilder;

    _customizedContentInput : CU00xDialogContent(THIS^);
END_VAR

VAR
    _dataLoadProcessSettings : BOOL;
    _dataLoadProcessSettingsByPlaner : BOOL;
    _dataCreateNew : BOOL;
    _dataOpen : BOOL;
    _dataClose : BOOL;
    _dataFinalize : BOOL;
    _continueRestore : BOOL;
    _loop : BOOL;
    _inspectionResult : BOOL;
    _inspectionDimensionResult : REAL;
    _tagsPairing : BOOL;
    _reqKey : STRING;
    _reqAssignedValue : STRING;
    _inspectorSingleExamples : BOOL;
    _inspectorGroupExamples : BOOL;
	_dialogExamples : BOOL;

END_VAR

Run();

(*~
	<docu>
		<summary>
			Loads technology settings from the current technology set into this controlled unit.
			The `StationProcessDataManager.Data` is populated by data from process settings.						
		</summary>
	</docu>
~*)
METHOD DataLoadProcessSettings : BOOL
VAR_INPUT
	inStepID : INT;
END_VAR

VAR
	_ans: TcoCore.eDialogAnswer;
END_VAR
IF (Step(inStepID, _dataLoadProcessSettings, 'LOAD PROCESS SETTING')) THEN
    //-------------------------------------
	
	THIS^._missingProcessSettingMessage.OnCondition(Station.Technology.ProcessSettings.Data._EntityId = '')
									   .Build()
									   .Append('No process data. Please load setting')
									   .As()				   
									   .AsError()
									   .Pin();
					   
				   
	IF(Station.Technology.ProcessSettings.Data._EntityId <> '' (*AND NOT THIS^._missingProcessSettingMessage.Pinned*)) THEN
		IF(Station.Technology.ProcessSettings.Read(Station.Technology.ProcessSettings.Data._EntityId).Done) THEN
			Station.ProcessDataManager.Data := Station.Technology.ProcessSettings.Data;
			Station.ProcessDataManager.Data.EntityHeader.RecipeCreated := Station.Technology.ProcessSettings.Data._Created;
			Station.ProcessDataManager.Data.EntityHeader.RecipeLastModified  := Station.Technology.ProcessSettings.Data._Modified;
			Station.ProcessDataManager.Data.EntityHeader.Recipe  := Station.Technology.ProcessSettings.Data._EntityId;				
			CompleteStep();

		END_IF;	
	ELSE
		_ans:=_dialog.Show()
			.WithImage('d:\MTS\Develop\TcOpenGroup\TcOpen\assets\logo\TcOpenWide.png',400,600)	
	       .WithCaption('<#Process data not selected#>')
		   .WithText('<#Would you like to load default settings?#>')
		   .WithYesNoCancel().Answer;
		IF(_ans=TcoCore.eDialogAnswer.Cancel) THEN
			this^.Restore();
		END_IF
		IF( _ans= TcoCore.eDialogAnswer.Yes) THEN
		   
		   	Station.Technology.ProcessSettings.Data._EntityId := 'default';
		END_IF; 

			
	END_IF		    				
    //-------------------------------------
END_IF
END_METHOD

(*~
	<docu>
		<summary>
			Loads process settings from the current process set into this controlled unit.
			The `StationProcessDataManager.Data` is populated by data from process settings.						
		</summary>
	</docu>
~*)
METHOD DataLoadProcessSettingsByPlaner : BOOL
VAR_INPUT
	inStepID : INT;
END_VAR
IF (Step(inStepID, _dataLoadProcessSettingsByPlaner, 'LOAD PROCESS SETTING BY THE PRODUCTION PLANER')) THEN
    //-------------------------------------


								   
	 IF Station.ProductionPlanerTask.Invoke().Done	AND_THEN(Station.ProductionPlanerTask.RequiredProcessSettingsId <> '') THEN
		
		IF NOT Station.ProductionPlanerTask.ProductionPlanCompleted and_then (Station.Technology.ProcessSettings.Read(Station.ProductionPlanerTask.RequiredProcessSettingsId).Done)
			 THEN
			Station.ProcessDataManager.Data := Station.Technology.ProcessSettings.Data;
			Station.ProcessDataManager.Data.EntityHeader.RecipeCreated := Station.Technology.ProcessSettings.Data._Created;
			Station.ProcessDataManager.Data.EntityHeader.RecipeLastModified  := Station.Technology.ProcessSettings.Data._Modified;
			Station.ProcessDataManager.Data.EntityHeader.Recipe  := Station.Technology.ProcessSettings.Data._EntityId;				
			CompleteStep();
			Station.ProductionPlanerTask.Restore();
		END_IF;
	ELSIF  Station.ProductionPlanerTask.ProductionPlanIsEmpty THEN
		IF (_dialog.Show()
	       .WithCaption('<#Production planer#>')
		   .WithText('<#Production planer is empty!#>')
			.WithOk().Answer = TcoCore.eDialogAnswer.OK) THEN;
			;// Production plan comleted , here you can write diferent scenario ( leave it with current state , provide ground etc)	 
	
		 	//Station.GroundTask.Task.Invoke();
		   
		End_if;
	
	ELSIF  Station.ProductionPlanerTask.ProductionPlanCompleted THEN
		IF (_dialog.Show()
	       .WithCaption('<#Production planer#>')
		   .WithText('<#Production planer completed required plan!#>')
			.WithOk().Answer = TcoCore.eDialogAnswer.OK) THEN;
			;// Production plan comleted , here you can write diferent scenario ( leave it with current state , provide ground etc)	 
	
		 	//Station.GroundTask.Task.Invoke();
		   
		End_if;

			
	END_IF		    				
    //-------------------------------------
END_IF
END_METHOD

(*~
	<docu>
		<summary>
			Wait for start operations and then go into this controlled unit sequence.						
		</summary>
	</docu>
~*)
METHOD DataReadyForOperations : BOOL
VAR_INPUT
	inStepID : INT;
END_VAR

VAR
	_ans: TcoCore.eDialogAnswer;
END_VAR
THIS^.Station.ResetReadyForOperations();   

IF (Step(inStepID, TRUE, '<#READY TO START OPERATIONS#>')) THEN
    //-------------------------------------
	
	THIS^.Station.SetReadyForOperations();   
	
  	Await(THIS^.Station.InternalRetrieveEntity(inCarrier:=2(*here comes info from carousel position*),refStorage:=Station.Technology.InternalStorage) 
			 AND_THEN THIS^.Station.DoesBelong() 
			 AND_THEN THIS^.Station.RunOperations(refGlobalTrigger:=Station.Technology.RunOperations)
			 AND_THEN THIS^.Station.InternalOpenEntity(inCarrier:=2(*here comes info from carousel position*),refStorage:=Station.Technology.InternalStorage,inoHeader:= THIS^.Station.CuProcessData.Header));
    //-------------------------------------
END_IF
END_METHOD

METHOD DialogExamples
VAR_INPUT
		inStepID : INT;
END_VAR
IF (Step(inStepID, TRUE, 'DIALOG EXAMPLE ')) THEN
//-------------------------------------
		_dialog.Show()
            .WithType(eDialogType.Question)
            .WithYesNo()
            .WithCaption('Hey')
            .WithText('Do we go ahead ');

        IF (_dialog.Answer = TcoCore.eDialogAnswer.Yes) THEN
            CompleteStep();
        END_IF;

        IF (_dialog.Answer = TcoCore.eDialogAnswer.No) THEN
            ;
        END_IF;

//-------------------------------------
END_IF;

IF (Step(inStepID+10, TRUE, 'DIALOG EXAMPLE WIT IMAGE')) THEN
//-------------------------------------
		_dialog.Show()
            .WithType(eDialogType.Question)
            .WithYesNo()
			.WithImage('D:\MTS\Develop\TcOpenGroup\TcOpen\assets\logo\TcOpenLogo.png',400,600)
            .WithCaption('Hey 1')
            .WithText('Do we go ahead ?');

        IF (_dialog.Answer = TcoCore.eDialogAnswer.Yes) THEN
            CompleteStep();
        END_IF;

        IF (_dialog.Answer = TcoCore.eDialogAnswer.No) THEN
            ;
        END_IF;

//-------------------------------------
END_IF;


IF (Step(inStepID+20, TRUE, 'DIALOG EXAMPLE WITH CLOSE FROM PLC')) THEN
//-------------------------------------
		_dialog.ShowWithExternalClose(inOkAnswerSignal:=FALSE , inYesAnswerSignal:= CurrentStep.Duration>T#2000MS, inNoAnswerSignal:= FALSE, inCancelAnswerSignal:= FALSE)
		    .WithType(eDialogType.Info)
            .WithYesNoCancel()
            .WithCaption('Hey')
            .WithText('Do you wana retry it? Yes answer will be set in 4 sec?');

        IF (_dialog.Answer = TcoCore.eDialogAnswer.Yes) THEN
            CompleteStep();
        END_IF;

      

//-------------------------------------
END_IF;

IF (Step(inStepID+30, TRUE, 'CUSTOMIZED DIALOG EXAMPLE WITH CLOSE FROM PLC ')) THEN
//-------------------------------------
			 _dialogCustomized.ShowWithExternalClose(inOption1AnswerSignal:=FALSE,inOption2AnswerSignal:=FALSE, inOption3AnswerSignal:=CurrentStep.Duration>T#4000MS,inOption4AnswerSignal:=FALSE)
            
            .WithOption1('This is Option1=>retry')
			  .WithOption2('This is Option2=>first step')
			    .WithOption3('This is Option3 =>continue and finish in 4s')
			.WithImage('D:\MTS\Develop\TcOpenGroup\TcOpen\assets\logo\TcOpenWide.png',500,500)
            .WithCaption('Hey')
            .WithText('What we are going to do.');
            
		
           
	
			IF (_dialogCustomized.Answer = TcoCore.eCustomizedDialogAnswer.Option3) THEN
				CompleteStep();
			END_IF;

//-------------------------------------
END_IF;

IF (Step(inStepID+40, TRUE, 'INPUT DIALOG EXAMPLE  REQURED FIELDS TO INPUT DATA')) THEN
//-------------------------------------
		_dialogWithInput.Show(refContent:=_customizedContentInput)
            .WithType(eDialogType.Question)
            .WithYesNo()
            .WithCaption('Hey wana set data')
            .WithText('Do you realy want to sent data to ....?');
                
		IF (_dialogWithInput.Answer = TcoCore.eInputDialogAnswer.Yes) THEN
				CompleteStep();
			//by yes or (ok) option data are confirmed and transfered to plc (_customizedContentInput)
		ELSIF (_dialogWithInput.Answer = TcoCore.eInputDialogAnswer.No) THEN
			// data in struct '_customizedContentInput' remains same as before
 		END_IF;
		

//-------------------------------------
END_IF;
IF (Step(inStepID+50, TRUE, 'INPUT DIALOG EXAMPLE WITH WEB CONTENT AND REQURED FIELDS TO INPUT DATA')) THEN
//-------------------------------------
		_dialogWithInput.Show(refContent:=_customizedContentInput)
            .WithType(eDialogType.Question)
            .WithOk()
			.WithImage('https://github.com/TcOpenGroup',400,600)
            .WithCaption('Hey wana set data')
            .WithText('Do you realy want to sent data to ....?');
			
                
		IF (_dialogWithInput.Answer = TcoCore.eInputDialogAnswer.OK) THEN
			CompleteStep();
			
		END_IF;

//-------------------------------------
END_IF;
END_METHOD

METHOD GroupedExample
VAR_INPUT
		inStepID : INT;
END_VAR
IF (Step(inStepID, TRUE, 'MULTI ANALOGUE INSPECTIONS PART 1 WITH WEB CONTENT')) THEN
//-------------------------------------
		Station.GroupInspection
		.WithCoordinator(THIS^)
		.Act();
		Station.GroupInspection.Inspect(Station.ProcessDataManager.Data.CU00x.Dim_Inspector_1.WithCoordinator(THIS^).Inspect(0));	
		Station.GroupInspection.Inspect(Station.ProcessDataManager.Data.CU00x.Dim_Inspector_2.WithCoordinator(THIS^).Inspect(0));	
		Station.GroupInspection.Inspect(Station.ProcessDataManager.Data.CU00x.Dim_Inspector_3.WithCoordinator(THIS^).Inspect(0));	
		Station.GroupInspection.Inspect(Station.ProcessDataManager.Data.CU00x.Dim_Inspector_4.WithCoordinator(THIS^).Inspect(0));	
		Station.GroupInspection.Inspect(Station.ProcessDataManager.Data.CU00x.Dim_Inspector_5.WithCoordinator(THIS^).Inspect(0));	
		Station.GroupInspection.Inspect(Station.ProcessDataManager.Data.CU00x.Dim_Inspector_6.WithCoordinator(THIS^).Inspect(1));	
		Station.GroupInspection.Inspect(Station.ProcessDataManager.Data.CU00x.Dim_Inspector_7.WithCoordinator(THIS^).Inspect(0));	
		Station.GroupInspection.Inspect(Station.ProcessDataManager.Data.CU00x.Dim_Inspector_8.WithCoordinator(THIS^).Inspect(0));	
		Station.GroupInspection.Inspect(Station.ProcessDataManager.Data.CU00x.Dim_Inspector_9.WithCoordinator(THIS^).Inspect(0));	
		Station.GroupInspection.Inspect(Station.ProcessDataManager.Data.CU00x.Dim_Inspector_10.WithCoordinator(THIS^).Inspect(0));	
	
		
		Station.GroupInspection.UpdateComprehensiveResult(Station.ProcessDataManager.Data.EntityHeader.Results)	
		.Instruct('Something is wrong 1')
		.InstructWithImage('https://github.com/TcOpenGroup/TcOpen/blob/dev/README.md',400,600)	
		.OnFail()
		.Dialog(inStepID+10);			
//-------------------------------------
END_IF;
IF (Step(inStepID+10, TRUE, 'MULTI ANALOGUE INSPECTIONS PART 2 WITH INSTRUCTION AND DESCRIPTION')) THEN
//-------------------------------------
		Station.GroupInspection
		.WithCoordinator(THIS^)
		.Act();
		Station.GroupInspection.Inspect(Station.ProcessDataManager.Data.CU00x.Dim_Inspector_11.WithCoordinator(THIS^).Inspect(0));	
		Station.GroupInspection.Inspect(Station.ProcessDataManager.Data.CU00x.Dim_Inspector_12.WithCoordinator(THIS^).Inspect(0));	
		Station.GroupInspection.Inspect(Station.ProcessDataManager.Data.CU00x.Dim_Inspector_13.WithCoordinator(THIS^).Inspect(0));	
		Station.GroupInspection.Inspect(Station.ProcessDataManager.Data.CU00x.Dim_Inspector_14.WithCoordinator(THIS^).Inspect(0));	
		Station.GroupInspection.Inspect(Station.ProcessDataManager.Data.CU00x.Dim_Inspector_15.WithCoordinator(THIS^).Inspect(0));	
		Station.GroupInspection.Inspect(Station.ProcessDataManager.Data.CU00x.Dim_Inspector_16.WithCoordinator(THIS^).Inspect(1));	
		Station.GroupInspection.Inspect(Station.ProcessDataManager.Data.CU00x.Dim_Inspector_17.WithCoordinator(THIS^).Inspect(0));	
		Station.GroupInspection.Inspect(Station.ProcessDataManager.Data.CU00x.Dim_Inspector_18.WithCoordinator(THIS^).Inspect(0));	
		Station.GroupInspection.Inspect(Station.ProcessDataManager.Data.CU00x.Dim_Inspector_19.WithCoordinator(THIS^).Inspect(0));	
		Station.GroupInspection.Inspect(Station.ProcessDataManager.Data.CU00x.Dim_Inspector_20.WithCoordinator(THIS^).Inspect(0));	
	
		
		Station.GroupInspection.UpdateComprehensiveResult(Station.ProcessDataManager.Data.EntityHeader.Results)	
		.WithDescription()
		.Instruct('Something is wrong 2')
		.OnFail()
		.Dialog(inStepID+20);			
//-------------------------------------
END_IF;

IF (Step(inStepID+20, TRUE, 'DONE')) THEN
//-------------------------------------
		CompleteStep();
//-------------------------------------
END_IF;
END_METHOD

(*~
	<docu>
		<summary>
			Main method of the sequener. Custom code needs to be placed here. The sequencer is executed by call of **Instance.Run()** method.
			This method is abstract, and it must be overridden in derived block.
		</summary>
	</docu>
~*)
METHOD PROTECTED Main : BOOL
(*

	OPENING DATA OPERATIONS
	Following methods provide process data manipulation for this controlled unit.
	Remove `IF` statement and comment or uncomment according to your need.
*)
// Loads process settings. 
// Typically used in the first station of the technology to load process settings that will be used trough out the production
IF (_dataLoadProcessSettings) THEN
    THIS^.DataLoadProcessSettings(100);
END_IF;

// Loads process settings via produciton planer. 
// Typically used in the first station of the technology to load process settings that will be used trough out the production 
// .......
IF (_dataLoadProcessSettingsByPlaner) THEN
    THIS^.DataLoadProcessSettingsByPlaner(110);
END_IF;

(*

		
		This step we would like to star cycle time (e.g. we want to exclude loading data from clean cycle time )		
*)
IF (Step(150, TRUE, '<#START MEASURE CT TRIGGER#>')) THEN
    //-------------------------------------    
    StartCleanCycleTime();
    StepCompleteWhen(TRUE);
    //-------------------------------------
END_IF

// Creates new data entity (new part/item) 
// Typically used in the first station of the technology to create new document/record to be persited in the repository.
// Sets the status of the entity to 'InProgress'
IF (_dataCreateNew) THEN
	IF (Step(160, TRUE, 'CREATE ENTIY ID')) THEN
		//-------------------------------------    
		Station.ProcessDataManager.Data._EntityId := ULINT_TO_STRING(Context.RealTimeClock.TickClock());
	
		StepCompleteWhen(Station.ProcessDataManager.Data._EntityId<>'');
		//-------------------------------------
	END_IF
    THIS^.DataEntityCreateNew(200, Station.ProcessDataManager.Data._EntityId, Header := Station.ProcessDataManager.Data.CU00x.Header);
END_IF;

// Populates the information in the data header of this controlled unit (operation start time stamp, user info, etc)
// Typically used prior to starting operation within a controlled unit.
IF (_dataOpen) THEN
    THIS^.DataEntityOpen(300,
        30000,
        Station.ProcessDataManager.Data._EntityId,
        Station.ProcessDataManager.Data.CU00x.Header);
END_IF;


// Handle user defined carier id
// Typically used in the first station of the technology to assign user defined carier ID  instead of raw unique id(RfidChip....)
IF (_tagsPairing) THEN
    THIS^.PairTag(400);
END_IF;
(*

		STEPS OF THE SEQUENCE
		Here we would place steps to perfom the operations of this controlled unit.

*)



IF (Step(900, TRUE, 'SINGLE INSPECTION')) THEN
    //-------------------------------------    
	Station.ProcessDataManager.Data.CU00x.BoltPresenceInspector.Data.FailureDescription:='BoltPresenceInspector error';
    Station.ProcessDataManager.Data.CU00x.BoltPresenceInspector.WithCoordinator(THIS^)
        .Inspect(_inspectionResult)
        .UpdateComprehensiveResult(Station.ProcessDataManager.Data.EntityHeader.Results)
        .OnFail().CarryOn();
    //-------------------------------------
END_IF

IF (Step(910, TRUE, 'SINGLE ANALOGUE INSPECTION')) THEN
    //-------------------------------------    
		Station.ProcessDataManager.Data.CU00x.BoltDimensionPresenceInspector.Data.FailureDescription:='BoltDimensionPresenceInspector error';

    Station.ProcessDataManager.Data.CU00x.BoltDimensionPresenceInspector.WithCoordinator(THIS^)
        .Inspect(_inspectionDimensionResult)
        .UpdateComprehensiveResult(Station.ProcessDataManager.Data.EntityHeader.Results)
        .OnFail().Dialog(300);
    //-------------------------------------
END_IF


//dialog usage examples
IF _dialogExamples THEN
	DialogExamples(1000);
END_IF;

//single inspexction usage
IF _inspectorSingleExamples THEN
	SingleExample(1100);
END_IF;

// grouped usage of isnpectors
IF _inspectorGroupExamples THEN
	GroupedExample(1200);
END_IF;


IF (Step(2000, true, 'START PARALELL TASK')) THEN
    //-------------------------------------    
    StepCompleteWhen(_paralellTask.Task.Invoke().Busy);
    //-------------------------------------
END_IF

(*

		RECOVERY STEPS
		This step and the following steps should bring the controlled unit in a state from which 
		the sequence can be safely restarted from the beginning of the this sequencer. 		
*)
IF (Step(RESTORE_STEP_ID, TRUE, 'FIRST RESTORE STEP')) THEN
    //-------------------------------------
    StepCompleteWhen(_continueRestore);
    //-------------------------------------	
END_IF

(*

		
		This step we would save cycle time value (e.g. we not include saving data into cycle time )
		
*)
IF (Step(2150, TRUE, 'STOP MEASURE CT TRIGGER')) THEN
    //-------------------------------------    
    StopCleanCycleTime();
    StepCompleteWhen(TRUE);
    //-------------------------------------
END_IF

(*

	CLOSING DATA OPERATIONS
	Following methods provide process data manipulation for this controlled unit.
	Comment or uncomment according to your need.
*)
// Populates the information in the data header of this controlled unit (operations end time stamp, user info, etc)
// Typically used after all steps within the controlled unit are completed.
IF (_dataClose) THEN
    THIS^.DataEntityClose(5000, eDataEntityInvokeType.InvokeAndWaitDone, Station.ProcessDataManager.Data.CU00x.Header);
END_IF;

// Populates the information in the data header of this controlled unit (operations end time stamp, user info, etc)
// Typically used after all operation on the technology are completed.
// Input parameter eDataEntityInvokeType.InvokeOnly is used for speed up cycle(TRUE)
IF (_dataFinalize) THEN
    THIS^.DataEntityFinalize(5500, eDataEntityInvokeType.InvokeOnly, Station.ProcessDataManager.Data.CU00x.Header);
END_IF;

IF (Step(10000, TRUE, 'WAIT FOR PARALELL TASK TO FINISH')) THEN
    //-------------------------------------
    StepCompleteWhen(_paralellTask.Task.Done);

    IF _paralellTask.Task.Done THEN
        _paralellTask.Restore();
    END_IF
    //-------------------------------------	
END_IF

IF (Step(20000, _dataClose, 'WAIT FOR IF DATA FINALIZE IS DONE')) THEN
    //-------------------------------------
    StepCompleteWhen(Station.UpdateEntityTask.Done);
    //-------------------------------------	
END_IF


//monitor if conseccutive failures occur during automatic cycle. System monitor two basic types like are arbitrary failure in seqence, or  same(equal) failure in sequence
//if Number of allowed recurring failure is 0 , monitoring is inactive.
//Recurring failures are based on ErrorCodes in TcoComprehensiveResult.
//If error code in Same recurring failure is empty string ,monitorig of failure is not performed.
//Error code in Arbitrary Recuring failure is irelevant.    
THIS^.MonitorAnyRecurringFailure(22000,THIS^.Station._settings.AnyRecurringFailure>0 , Station.ProcessDataManager.Data.EntityHeader.Results);
THIS^.MonitorSameRecurringFailure(22100,THIS^.Station._settings.SameRecurringFailure>0 , Station.ProcessDataManager.Data.EntityHeader.Results);



IF (Step(30000, TRUE, 'LAST STEP')) THEN
    //-------------------------------------
    IF (_loop) THEN
        CompleteSequence();
    END_IF;
    //-------------------------------------	
END_IF

_paralellTask();
END_METHOD

METHOD PUBLIC OnStart
SUPER^.OnStart();
Station.GroundTask.Restore();
Station.ManualTask.Restore();
Station.GroundTask.CancelGround();
_paralellTask.Restore();
END_METHOD

(*~
	<docu>
		<summary>
			Loads process settings from the current process set into this controlled unit.
			The `StationProcessDataManager.Data` is populated by data from process settings.						
		</summary>
	</docu>
~*)
METHOD PairTag : BOOL
VAR_INPUT
	inStepID : INT;
END_VAR

VAR
	answer: TagsPairing;
	_addNewTag: BOOL;
	dialogAnswer: eDialogAnswer;
END_VAR
IF (Step(inStepID, _tagsPairing, '<#PAIR TAG WITH ASSIGNED VALUE EXAMPLE#>')) THEN
    //-------------------------------------
	_addNewTag:=FALSE;

	answer:= Station.Components.PairTagTask.Answer;
	//this field may be assigned by unique ID of rfid chip , or dmc code.The PairTagTask provide answer where is assigned user defined value for this unique ID value.
	//If not, there may be diferent scenarios defined. See example bellow.
	_reqKey:='123456789';				   
	 IF Station.Components.PairTagTask.Run(inMode:=eTagPairingMode.GetTag, inKey:=_reqKey ,inAssignedValue:='').Invoke().Done	 THEN
		
		IF  answer.Answer =eTagPairingAnswer.TagFound 
			 THEN
			Station.ProcessDataManager.Data.EntityHeader.Carrier := answer.AssignedValue;
			CompleteStep();
			Station.Components.PairTagTask.Restore();
		
		ELSIF  answer.Answer = eTagPairingAnswer.TagFoundInactive THEN
			IF (_dialog.Show()
			   .WithCaption('<#Pairing Tag#>')
			   .WithText(_sb.Clear().Append('<#Founded tag#> ').Append(_reqKey).Append(' <#is inactive!#> ').Append(Station.Components.PairTagTask.AnswerInstruction).ToString() )
				.WithOk().Answer = TcoCore.eDialogAnswer.OK) THEN;
				;// Founded tag is Inactive. Probably carier(pallete) was disasbled due produced many errors.Se  here you can write diferent scenario ( leave it with current state , provide ground etc)	 
		
				//Station.GroundTask.Task.Invoke();
			   
			End_if;
		
		ELSIF  answer.Answer = eTagPairingAnswer.TagFoundAssignedValueEmpty THEN
			  IF (_dialog.Show()
			   .WithCaption('<#Pairing Tag#>')
			   .WithText(_sb.Clear().Append('<#Tag#> ').Append(_reqKey).Append(' <#is founded but assigned value is empty! Would you like continue?#> ').Append(Station.Components.PairTagTask.AnswerInstruction).ToString() )
				.WithYesNo().Answer = TcoCore.eDialogAnswer.Yes) THEN;
				CompleteStep();
				Station.Components.PairTagTask.Restore();
			END_IF;
		   
		ELSIF  answer.Answer = eTagPairingAnswer.TagNotFound THEN
			  IF (_dialog.Show()
			   .WithCaption('<#Pairing Tag#>')
			   .WithText(_sb.Clear().Append('<#Tag#> ').Append(_reqKey).Append(' <#is not founded ! Would you like assign right now?#> ').Append(Station.Components.PairTagTask.AnswerInstruction).ToString() )
				.WithYesNo().Answer = TcoCore.eDialogAnswer.Yes) THEN;
				_addNewTag:=TRUE;
				CompleteStep();
				Station.Components.PairTagTask.Restore();
			END_IF;
	
		
			ELSIF  answer.Answer = eTagPairingAnswer.EmptyCollection THEN
			  IF (_dialog.Show()
			   .WithCaption('<#Pairing Tag#>')
			   .WithText(_sb.Clear().Append('<#Tag#> ').Append(_reqKey).Append(' <#is not founded due collection is empty ! Would you like assign right now?#> ').Append(Station.Components.PairTagTask.AnswerInstruction).ToString() )
				.WithYesNo().Answer = TcoCore.eDialogAnswer.Yes) THEN;
				_addNewTag:=TRUE;
				CompleteStep();
				Station.Components.PairTagTask.Restore();
			END_IF;
		End_if;
			
	END_IF		    				
    //-------------------------------------
END_IF

IF (Step(inStepID+10, _tagsPairing AND _addNewTag, '<#ADD NEW TAG  EXAMPLE#>')) THEN
    //-------------------------------------
	
	answer:= Station.Components.PairTagTask.Answer;
	//this field may be assigned by unique ID of rfid chip , or dmc code.The PairTagTask provide answer where is assigned user defined value for this unique ID value.
	//If not, there may be diferent scenarios defined. See example bellow.
	_reqKey:='123456789';		
	_reqAssignedValue := 'CustomIdExample123';	   
	 IF Station.Components.PairTagTask.Run(inMode:=eTagPairingMode.AddTag, inKey:=_reqKey, inAssignedValue:=_reqAssignedValue).Invoke().Done	 THEN
		
		IF  answer.Answer =eTagPairingAnswer.TagAddedSuccessfully 
			 THEN
			Station.ProcessDataManager.Data.EntityHeader.Carrier := answer.AssignedValue;
			CompleteStep();
			Station.Components.PairTagTask.Restore();
		END_IF;
	ELSIF  answer.Answer = eTagPairingAnswer.TagAlreadyExist THEN
		IF (_dialog.Show()
	       .WithCaption('<#Adding Tag#>')
		   .WithText(_sb.Clear().Append('<#Tag#> ').Append(_reqKey).Append(' <#already exist!#> ').Append(Station.Components.PairTagTask.AnswerInstruction).ToString() )
			.WithOk().Answer = TcoCore.eDialogAnswer.OK) THEN;
			;// Founded tag is Inactive. Probably carier(pallete) was disasbled due produced many errors.Se  here you can write diferent scenario ( leave it with current state , provide ground etc)	 
	
		 	//Station.GroundTask.Task.Invoke();
		   
		End_if;
	
	ELSIF  answer.Answer = eTagPairingAnswer.TagAddedNotSuccessfuly THEN
			dialogAnswer := _dialog.Show()
	       .WithCaption('<#Pairing Tag#>')
		   .WithText(_sb.Clear().Append('<#Tag#> ').Append(_reqKey).Append(' <#was not founnd! Would you like still like to continue?#> ').Append(Station.Components.PairTagTask.AnswerInstruction).ToString() )
			.WithYesNo().Answer;
			
	      IF (dialogAnswer= TcoCore.eDialogAnswer.Yes) THEN;
			CompleteStep();
			Station.Components.PairTagTask.Restore();
		END_IF;
		   

			
	END_IF		    				
    //-------------------------------------
END_IF
END_METHOD

METHOD SingleExample : BOOL
VAR_INPUT
		inStepID : INT;
END_VAR

IF (Step(inStepID, TRUE, 'SINGLE INSPECTION')) THEN
    //-------------------------------------    
	Station.ProcessDataManager.Data.CU00x.BoltPresenceInspector.Data.FailureDescription:='BoltPresenceInspector error';
    Station.ProcessDataManager.Data.CU00x.BoltPresenceInspector.WithCoordinator(THIS^)
        .Inspect(_inspectionResult)
        .UpdateComprehensiveResult(Station.ProcessDataManager.Data.EntityHeader.Results)
        .OnFail().Dialog(inStepID+10);
    //-------------------------------------
END_IF

// with checking if specific inspector is overinspected
IF (Step(inStepID+10, TRUE, 'SINGLE ANALOGUE INSPECTION')) THEN
//-------------------------------------
	Station.ProcessDataManager.Data.CU00x.BoltDimensionPresenceInspector.Data.FailureDescription:='BoltDimensionPresenceInspector error';
	Station.ProcessDataManager.Data.CU00x.BoltDimensionPresenceInspector.Data.NumberOfAllowedRetries:=100;
	IF NOT Station.ProcessDataManager.Data.CU00x.BoltDimensionPresenceInspector.OverInspected THEN
	
		Station.ProcessDataManager.Data.CU00x.BoltDimensionPresenceInspector.WithCoordinator(THIS^)
			.Inspect(_inspectionDimensionResult)
			.WithDescription()
			.UpdateComprehensiveResult(Station.ProcessDataManager.Data.EntityHeader.Results)
			.OnFail().Retry(inStepID+20);
	ELSE
	 	RequestStep(RESTORE_STEP_ID);	
	END_IF
//-------------------------------------
END_IF;

IF (Step(inStepID+20, TRUE, 'DONE')) THEN
//-------------------------------------
		CompleteStep();
//-------------------------------------
END_IF;
END_METHOD

PROPERTY Station : REFERENCE TO CU00x
GET
VAR
    _station : POINTER TO CU00x;
END_VAR
IF __QUERYPOINTER(Parent, _station) THEN // Check if _Parent is Station001
    Station REF= _station^;              // If the check is successful dereference a pointer. simlar to THIS^ or SUPER^
END_IF
END_GET
END_PROPERTY

END_FUNCTION_BLOCK

// ---- Abstractions/CUBase/Tasks/CUBaseAutomat.TcPOU
FUNCTION_BLOCK ABSTRACT CUBaseAutomat EXTENDS TcoTaskedSequencer
VAR
    _dialog : TcoCore.TcoDialog(THIS^);
    _dialogCustomized : TcoCore.TcoCustomizedDialog(THIS^);
    _dialogWithInput : TcoCore.TcoInputDialog(THIS^);
    {attribute addProperty Name "<#Clear counter#>"}
    _counterDataClear : TcoCore.TcoTask(THIS^);
END_VAR
VAR PERSISTENT
    _counterData : BasicCounterData := (Parent := THIS^);
END_VAR

METHOD PUBLIC ClearCounter
VAR_INPUT
END_VAR
_counterData.Passed := 0;
_counterData.Failed := 0;


_counterData.Total := _counterData.Passed + _counterData.Failed;
END_METHOD

PROPERTY PUBLIC ClearCounterDataTask : REFERENCE TO TcoCore.TcoTask
GET
ClearCounterDataTask ref=_counterDataClear;
END_GET
END_PROPERTY

METHOD Count
VAR_INPUT
	Header 		: EntityHeader;
	
END_VAR


IF NOT Header.IsEmpty THEN

    _counterData.LifeTime := _counterData.LifeTime + 1;

    IF Header.Results.Result = eOverallResult.Failed THEN
        _counterData.Failed := _counterData.Failed + 1;
        _counterData.LifeTimeFailed := _counterData.LifeTimeFailed + 1;
    ELSE
        _counterData.Passed := _counterData.Passed + 1;
        _counterData.LifeTimePassed := _counterData.LifeTimePassed + 1;
    END_IF

END_IF;

_counterData.Total := _counterData.Passed + _counterData.Failed;
END_METHOD

(*~
	<docu>
		<summary>
			Stores the data from this controlled unit into the repository. In addition modifies entity header and controlled unit header.									
		</summary>
	</docu>
~*)
METHOD DataEntityClose
VAR_INPUT
	(*~
	<docu>
		<summary>
			The unique step id definition.
		</summary>			
	</docu>	
	~*)
	inStepID : INT;
	(*~
	<docu>
		<summary>
			If input enum is set to InvokeAndWaitDone  operation will  wait until task reaches the ```Done``` state .
			If input enum is set to InvokeOnly results return True when  task reaches the ```Busy``` state . Later is recomended (neccessary) to check  task  ```Done``` state  , check  task  status.
		</summary>			
	</docu>	
	~*)
	InvokeAction: eDataEntityInvokeType;
END_VAR
VAR_IN_OUT
	Header : CuHeader; 
END_VAR
IF (Step(inStepID,TRUE, 'CLOSE ENTITY DATA')) THEN
    //-------------------------------------		
	IF IsFreshState THEN
		Count(THIS^.StationBase.ProcessDataManager.Data.EntityHeader);
	END_IF
	CASE InvokeAction OF
		eDataEntityInvokeType.InvokeAndWaitDone: 
				StepCompleteWhen(THIS^.StationBase.EntityFlowCloseForOperations(Header).Done);
		eDataEntityInvokeType.InvokeOnly: 
				StepCompleteWhen(THIS^.StationBase.EntityFlowCloseForOperations(Header).Busy);	
	END_CASE;			   		    				
    //-------------------------------------
END_IF
END_METHOD

(*~
	<docu>
		<summary>
			Creates new record in the repository with given EntityId and populates with the current controlled units data.
			In addition modifies entity header and controlled unit header.									
		</summary>
	</docu>
~*)
METHOD DataEntityCreateNew
VAR_INPUT	
	inStepID : INT;
	EntityId : STRING(255);
END_VAR

VAR_IN_OUT
	Header: CuHeader;
END_VAR
IF (Step(inStepID, TRUE, 'CREATE NEW ENTITY DATA')) THEN
    //-------------------------------------		
	StepCompleteWhen(THIS^.StationBase.EntityFlowCreateNew(EntityId, Header).Done);				   		    				
    //-------------------------------------
END_IF
END_METHOD

METHOD DataEntityDiscard
VAR_INPUT	
	inStepID : INT;
	EntityId : STRING(255);
END_VAR
VAR_IN_OUT
	Header: CuHeader;
END_VAR
IF (Step(inStepID, TRUE, 'DISCARD ENTITY DATA')) THEN
    //-------------------------------------		
	StepCompleteWhen(THIS^.StationBase.EntityFlowDiscard(EntityId, Header).Done);				   		    				
    //-------------------------------------
END_IF
END_METHOD

(*~
	<docu>
		<summary>
			Stores data of this controlled unit into the repository.
			In addition modifies entity header and controlled unit header.
			Finalize will set the comprehensive result from InProgress to Passed. 
			If the comprehensive result is Failed the finalizing will not modify the result.									
		</summary>
	</docu>
~*)
METHOD DataEntityFinalize : BOOL
VAR_INPUT
	(*~
	<docu>
		<summary>
			The unique step id definition.
		</summary>			
	</docu>	
	~*)
	inStepID : INT;
	(*~
	<docu>
		<summary>
			If input enum is set to InvokeAndWaitDone  operation will  wait until task reaches the ```Done``` state .
			If input enum is set to InvokeOnly results return True when  task reaches the ```Busy``` state . This option is used when we need to reduce cycle time. Later is recomended (neccessary) to check  task  ```Done``` state  , check  task  status.
		</summary>			
	</docu>	
	~*)
	InvokeAction: eDataEntityInvokeType;
END_VAR
VAR_IN_OUT
	Header: CuHeader;
END_VAR
IF (Step(inStepID,TRUE, 'FINALIZE ENTITY DATA')) THEN
    //-------------------------------------		
		CASE InvokeAction OF
		eDataEntityInvokeType.InvokeAndWaitDone: 
				StepCompleteWhen(THIS^.StationBase.EntityFlowFinalize(Header).Done);
		eDataEntityInvokeType.InvokeOnly: 
				StepCompleteWhen(THIS^.StationBase.EntityFlowFinalize(Header).Busy);	
	END_CASE;			   		    				
	StepCompleteWhen(THIS^.StationBase.EntityFlowFinalize(Header).Done );				   		    				
    //-------------------------------------
END_IF
END_METHOD

(*~
	<docu>
		<summary>
			Retrieves the data with given EntityId from the repository. In addition modifies entity header and controlled unit header.									
		</summary>
	</docu>
~*)
METHOD DataEntityOpen
VAR_INPUT
	(*~
	<docu>
		<summary>
			The unique step id definition.
		</summary>			
	</docu>	
	~*)
	inStepID : INT;
	(*~
	<docu>
		<summary>
			The definition of jump sptep.Usage of this jump step is when entity does not belong to the Controled unit.
		</summary>			
	</docu>	
	~*)
	inReqStepId: INT;
	inEntityId : STRING(255);
END_VAR
VAR_IN_OUT
	CuHeader: CuHeader;
END_VAR
IF (Step(inStepID, TRUE, 'OPEN ENTITY DATA')) THEN
    //-------------------------------------		
    IF THIS^.StationBase.EntityFlowOpenForOperations(inEntityId, CuHeader).Done THEN
        IF THIS^.StationBase.ProcessDataManager.Data.EntityHeader.IsEmpty THEN
            RequestStep(inReqStepId);
        ELSIF EntityDoesBelong() THEN
            CompleteStep();
        ELSE
            RequestStep(inReqStepId);
        END_IF
    END_IF;
    //-------------------------------------
END_IF
END_METHOD

METHOD EntityDoesBelong : BOOL
VAR_INPUT
END_VAR
EntityDoesBelong:=THIS^.StationBase.ProcessDataManager.Data.EntityHeader.NextStation = THIS^.StationBase.CuId;
END_METHOD

METHOD PUBLIC  HideAllDialogs
VAR_INPUT
END_VAR
_dialog.Restore();
_dialogWithInput.Restore();
_dialogCustomized.Restore();
END_METHOD

METHOD MonitorAnyRecurringFailure
VAR_INPUT
	(*~
	<docu>
		<summary>
			The unique step id definition.
		</summary>			
	</docu>	
	~*)
	inStepID : INT;
	(*~
	<docu>
		<summary>
			The step enable condition.
		</summary>			
	</docu>	
	~*)
	inEnableStep :BOOL;
	inResult : TcoComprehensiveResult;
END_VAR
IF (Step(inStepID,inEnableStep, 'MONITOR ANY RECURRING FAILURE IN SEQUENCE')) THEN
    //-------------------------------------		
	
	IF(inResult.Result<>eOverallResult.Failed ) THEN
		THIS^.StationBase.RecurringFails.AnyRecurringFails.Counter:=0;
		THIS^.StationBase.RecurringFails.AnyRecurringFails.Reached :=FALSE;
		This^.CompleteStep();
	ELSE
		//collect any recurring fails
		IF NOT THIS^.StationBase.RecurringFails.AnyRecurringFails.Reached THEN 
			THIS^.StationBase.RecurringFails.AnyRecurringFails.Counter := THIS^.StationBase.RecurringFails.AnyRecurringFails.Counter +1;
		END_IF
		THIS^.StationBase.RecurringFails.AnyRecurringFails.Reached:=THIS^.StationBase.RecurringFails.AnyRecurringFails.Counter>=THIS^.StationBase._settings.AnyRecurringFailure;
		

		
	

		
		THIS^.Messenger.OnCondition(THIS^.StationBase.RecurringFails.AnyRecurringFails.Reached)
									   .Build()
									   .Append('(Consecutive failure) The number of any recurring failure count has been reached!')
									   .Append(' Failure code: ')
									   .Append(inResult.ErrorCodes)
  									   .Append(' ')
									   .Append(inResult.Failures)						
									   .As()				   
									   .AsError();
									   
		THIS^.StepCompleteWhen(NOT THIS^.StationBase.RecurringFails.AnyRecurringFails.Reached);			
						   
									   
		IF THIS^.StationBase.RecurringFails.AnyRecurringFails.Reached THEN
			
				
			IF(_dialog.Show()
			   .WithCaption('<#(Consecutive failure) The number of any recurring failure count has been reached!#>')
			   .WithText('<#Please acknowledge recurring failure!#>')
			   .WithOk().Answer = TcoCore.eDialogAnswer.OK) THEN
			   
					THIS^.StationBase.RecurringFails.AnyRecurringFails.Counter:=0;
					THIS^.StationBase.RecurringFails.AnyRecurringFails.Reached :=FALSE;
					THIS^.CompleteStep();
			END_IF; 
		END_IF;
	END_IF;
	

	
	
	
 		    				
    //-------------------------------------
END_IF
END_METHOD

METHOD MonitorSameRecurringFailure
VAR_INPUT
	(*~
	<docu>
		<summary>
			The unique step id definition.
		</summary>			
	</docu>	
	~*)
	inStepID : INT;
		(*~
	<docu>
		<summary>
			The step enable condition.
		</summary>			
	</docu>	
	~*)
	inEnableStep :BOOL;
	inResult : TcoComprehensiveResult;
END_VAR
IF (Step(inStepID,inEnableStep, 'MONITOR SAME RECURRING FAILURE IN SEQUENCE')) THEN
    //-------------------------------------		
	
	IF(inResult.Result<>eOverallResult.Failed ) THEN
		THIS^.StationBase.RecurringFails.SameRecurringFails.Counter:=0;
		THIS^.StationBase.RecurringFails.SameRecurringFails.Reached :=FALSE;
		THIS^.CompleteStep();
	ELSE
	
		//collect same recurring
		IF NOT THIS^.StationBase.RecurringFails.SameRecurringFails.Reached THEN 
			IF THIS^.StationBase.RecurringFails.SameRecurringFails.Result.ErrorCodes = inResult.ErrorCodes AND inResult.ErrorCodes <>';' THEN //if error code not defined ignore
				THIS^.StationBase.RecurringFails.SameRecurringFails.Counter := THIS^.StationBase.RecurringFails.SameRecurringFails.Counter +1;
			END_IF;
			THIS^.StationBase.RecurringFails.SameRecurringFails.Result.ErrorCodes := inResult.ErrorCodes ;
		END_IF;
		
		THIS^.StationBase.RecurringFails.SameRecurringFails.Reached:=THIS^.StationBase.RecurringFails.SameRecurringFails.Counter>=THIS^.StationBase._settings.SameRecurringFailure;

			
		THIS^.Messenger.OnCondition(THIS^.StationBase.RecurringFails.SameRecurringFails.Reached)
									   .Build()
									   .Append('(Consecutive failure) The number of same recurring failure count has been reached!')
									   .Append(' Failure code: ')
									   .Append(inResult.ErrorCodes)
  									   .Append(' ')
									   .Append(inResult.Failures)									   									   
									   .As()				   
									   .AsError();
		
		THIS^.StepCompleteWhen(NOT THIS^.StationBase.RecurringFails.SameRecurringFails.Reached);
	

									   
		IF THIS^.StationBase.RecurringFails.SameRecurringFails.Reached THEN
			IF(_dialog.Show()
			   .WithCaption('<#(Consecutive failure) The number of same recurring failure count has been reached!#>')
			   .WithText('<#Please acknowledge recurring failure!#>')
			   .WithOk().Answer = TcoCore.eDialogAnswer.Ok) THEN
			   
					THIS^.StationBase.RecurringFails.SameRecurringFails.Counter:=0;
					THIS^.StationBase.RecurringFails.SameRecurringFails.Reached :=FALSE;
					THIS^.CompleteStep();
			END_IF; 
		END_IF
	END_IF;
	

	
	
	
 		    				
    //-------------------------------------
END_IF
END_METHOD

PROPERTY StationBase : REFERENCE TO CuBase
GET
VAR
    _station : POINTER TO CUBase;
END_VAR
IF __QUERYPOINTER(Parent, _station) THEN // Check if _Parent is Station001
    StationBase REF= _station^;              // If the check is successful dereference a pointer. simlar to THIS^ or SUPER^
END_IF
END_GET
END_PROPERTY

END_FUNCTION_BLOCK

// ---- Abstractions/TcoCore/TcoTaskedSequencer.TcPOU
FUNCTION_BLOCK PUBLIC ABSTRACT TcoTaskedSequencer EXTENDS TcoCore.TcoSequencerBase
VAR
	{attribute addProperty Name "|[[1]AttributeName]|"}
	{attribute addProperty ToolTip "|[[1]AttributeToolTip]|"}
    _task : TcoInnerTask(THIS^);
    _o    : TcoCore.TcoSequencerObserver(THIS^);	
	{attribute addProperty Name "|[[1]Cycle Time Analitics]|"} 
	_cycleTimeAnalitics:CycleTimeAnalitics;	
	_startCleanCycleTime: TIME;
	_stopCleanCycleTime: TIME;
	_timer_1: TON;
	_timer_2: TON;
	_suspenStepExecution:BOOL;
END_VAR

Run();

PROPERTY PUBLIC AverageCleanCycleTime : TIME
GET
AverageCleanCycleTime:=_cycleTimeAnalitics.AverageCleanCycle;
END_GET
END_PROPERTY

PROPERTY PUBLIC AverageCycleTime : TIME
GET
AverageCycleTime:=_cycleTimeAnalitics.Average;
END_GET
END_PROPERTY

(*~
	<docu>
		<summary>
			Completes the actually running step, when the `inCondition` parameter is `TRUE`.
			Method is typically called inside a step as the transition method.
		</summary>			
	</docu>	
~*)
METHOD PROTECTED FINAL Await
VAR_INPUT
    (*~
	<docu>
		<summary>
			The condition under which the step is completed.
		</summary>			
	</docu>	
~*)
    inCondition : BOOL;
END_VAR
i_StepCompleteWhen(inCondition := inCondition);
END_METHOD

(*~
	<docu>
		<summary>
			<para>
				Completes the sequencer, and return the sequencer pointer to the first step in the seuqence.
				Method is typically called inside the last step of the sequence.
			</para>
		</summary>			
	</docu>	
~*)
METHOD PROTECTED FINAL CompleteSequence
i_CompleteSequence();

IF _cycleTimeAnalitics.FilterConstant = 0 THEN;
	_cycleTimeAnalitics.FilterConstant:=10;
END_IF;


IF _cycleTimeAnalitics.Average = T#0S THEN
	_cycleTimeAnalitics.Average:=_SequenceElapsedTime;
END_IF
_cycleTimeAnalitics.Average:= (((_cycleTimeAnalitics.FilterConstant-1)*_cycleTimeAnalitics.Average)+_LastCycleTime)/_cycleTimeAnalitics.FilterConstant;

_startCleanCycleTime:=T#0S;
_stopCleanCycleTime:=T#0S;
END_METHOD

(*~
	<docu>
		<summary>
			Completes the execution of the current step and moves the sequencer pointer to the next step in order of execution.
			The call returns `ITcoObjectRestorer` that allows to restore object upon step completition.
		</summary>		
		<returns></returns>	
	</docu>	
~*)
METHOD PROTECTED FINAL CompleteStep : ITcoObjectRestorer
CompleteStep := i_CompleteStep();
END_METHOD

PROPERTY PUBLIC CycleTimeFilterConstant : UINT
GET
CycleTimeFilterConstant:=_cycleTimeAnalitics.FilterConstant;
END_GET
SET // PUBLIC
_cycleTimeAnalitics.FilterConstant:=CycleTimeFilterConstant;
END_SET
END_PROPERTY

(*~
	<docu>
		<summary>
			Main method of the sequener. Custom code needs to be placed here. The sequencer is executed by call of **Instance.Run()** method.
			This method is abstract, and it must be overridden in derived block.
		</summary>
	</docu>
~*)
METHOD PROTECTED  Main : BOOL
END_METHOD

(*~
	<docu>
		<summary>
			Completes the execution of the current step and moves the sequencer pointer to the next step in order of execution.
			The call returns `ITcoObjectRestorer` that allows to restore object upon step completition.
		</summary>		
		<returns></returns>	
	</docu>	
~*)
METHOD PROTECTED FINAL Next : ITcoObjectRestorer
Next := i_CompleteStep();
END_METHOD

METHOD PUBLIC OnAbort : BOOL
SUPER^.Restore();
END_METHOD

METHOD PUBLIC OnDone : BOOL
END_METHOD

METHOD PUBLIC OnError : BOOL
END_METHOD

METHOD PUBLIC OnStart
_startCleanCycleTime:=T#0S;
_stopCleanCycleTime:=T#0S;
END_METHOD

METHOD pr_Close
VAR_INPUT
END_VAR
_lastClosingCycle := Context.StartCycleCount;

IF _sequencerHasError THEN
    OnSequencerError(_sequencerErrorId);
END_IF

_previousNumberOfStepsInSequence := _numberOfStepsInSequence;
Context.Environment.Messaging.Suspend();

IF _modeController._stepIn.Done THEN
    _modeController._stepIn.Restore();
END_IF

Context.Environment.Messaging.Resume();

_restoringSequence := FALSE;
END_METHOD

METHOD pr_Open
VAR
    _message : STRING(255);
END_VAR
_theOrderOfTheCurrentlyEvaluatedStep := 0;

IF _requestStepActive AND
    _requestedStepId <> (MinStepID - 1) AND
    (_modeController.Mode <> eSequencerMode.StepMode OR _modeController._stepIn.Busy OR _checkStepIdRequestedInStepMode) THEN
    _requestStepCycle := _requestStepCycle + 1;
ELSE
    _requestStepCycle := 0;
END_IF

IF _requestStepCycle > 1 AND NOT _sequencerHasError THEN
    _sequencerErrorId        := eSequencerError.StepWithRequestedIdDoesNotExists;
    _message                 := CONCAT('REQUESTED STEP_ID: ', INT_TO_STRING(_requestedStepId));
    _message                 := CONCAT(_message, ' DOES NOT EXIST');
    _currentStep.Description := _message;
    _currentStep.Status      := eStepStatus.Error;
    THIS^.Messenger.Post(_message, eMessageCategory.ProgrammingError);
    _sequencerHasError := TRUE;
END_IF

IF _StepIdUniquenessControlState = eStepIdUniquenessControlState.NotYetStarted OR
    _StepIdUniquenessControlState = eStepIdUniquenessControlState.Requested THEN
    _StepIdUniquenessControlState := eStepIdUniquenessControlState.Started;
END_IF;

_restoringSequence := FALSE;

_lastOpeningCycle := Context.StartCycleCount;
;
END_METHOD

(*~
	<docu>
		<summary>
			Terminates the currently executed step and set the sequencer's pointer to the step with Id that corresponds to ```inRequestedStepID``` parameter.
			When the order of the requested step is higher than the order of the currently finished step (the requested step is "after" the current one)
			the requested step is started in the same context cycle.
			When the order of the requested step is lower than the order of the currently finished step (the requested step is "before" the current one)
			the requested step is started in the next context cycle.
			If the requested step is not found even in the next context cycle, the sequencer enters error state ```StepWithRequestedIdDoesNotExists```.
			<para>
				See <see cref="TcoCore.eSequencerError"/> for detailed description.
			</para>
		</summary>
	</docu>
~*)
METHOD PROTECTED FINAL RequestRestoreOrigin : ITcoSequencer

VAR
    _message : STRING(254);
END_VAR
RequestRestoreOrigin := i_RequestStep(inRequestedStepID := RESTORE_STEP_ID);
END_METHOD

(*~
	<docu>
		<summary>
			Terminates the currently executed step and set the sequencer's pointer to the step with Id that corresponds to ```inRequestedStepID``` parameter.
			When the order of the requested step is higher than the order of the currently finished step (the requested step is "after" the current one)
			the requested step is started in the same context cycle.
			When the order of the requested step is lower than the order of the currently finished step (the requested step is "before" the current one)
			the requested step is started in the next context cycle.
			If the requested step is not found even in the next context cycle, the sequencer enters error state ```StepWithRequestedIdDoesNotExists```.
			<para>
				See <see cref="TcoCore.eSequencerError"/> for detailed description.
			</para>
		</summary>
	</docu>
~*)
METHOD PROTECTED FINAL RequestStep : ITcoSequencer
VAR_INPUT
    (*~
		<docu>
			<summary>
				StepId of the step to be executed.
			</summary>
		</docu>
	~*)
    inRequestedStepID : INT := MinStepID - 1;
END_VAR
VAR
    _message : STRING(254);
END_VAR
RequestStep := i_RequestStep(inRequestedStepID := inRequestedStepID);
END_METHOD

(*~
	<docu>
		<summary>
			This method resets the sequencer cycle time . 
				Method is typically called before starting the sequence(e.g.in ground position task) .
		</summary>		
		<returns></returns>	
	</docu>	
~*)
METHOD PUBLIC ResetCycleTime
VAR_INPUT
END_VAR

_cycleTimeAnalitics.Average:=T#0S;
_cycleTimeAnalitics.AverageCleanCycle:=T#0S;
END_METHOD

METHOD PRIVATE ResetTimers
VAR_INPUT
END_VAR
_timer_1.IN:=FALSE;
_timer_2.IN:=FALSE;
END_METHOD

(*~
	<docu>
		<summary>
			<para>
				This method resets the sequencer. 
				Method is typically called before starting the sequence or after error has occured in the sequence.
			</para>
		</summary>			
	</docu>	
~*)
METHOD PUBLIC Restore : ITcoRestorable
SUPER^.Restore();
Task.Restore();
_suspenStepExecution:=false;
END_METHOD

(*~
	<docu>
		<summary>
			<para>
				Ensures calling the Open(), Main() and Close() methods in the desired order.
				This method is final, so it cannot be overloaded. The **Instance.Run()** needs to be called cyclically inside the appropriate context.
			</para>
		</summary>			
	</docu>	
~*)
METHOD PUBLIC FINAL Run
VAR
    _message : STRING;
END_VAR
IF (_task.Execute()) THEN
    THIS^.pr_Open();
    THIS^.Observer := _o;
    THIS^.Main();
    THIS^.pr_Close();
END_IF;
END_METHOD

(*~
	<docu>
		<summary>
			This method s used to start the clean cycle time measurement . 
				Method is typically called at the beggining of the sequence(e.g.in automat sequence) .
		</summary>		
		<returns></returns>	
	</docu>	
~*)

METHOD PUBLIC StartCleanCycleTime
VAR_INPUT
END_VAR
_stopCleanCycleTime:=t#0s;
_startCleanCycleTime:=_SequenceElapsedTime;
END_METHOD

METHOD PROTECTED Step : BOOL
VAR_INPUT
    (*~
	<docu>
		<summary>
			StepId of the current step.
			<remarks>			
				<note type="important">
					This number must be unique throughout the complete sequence.
					It must be a constant or numerical literal and it must not change during the life-time of the sequencer. 
				</note>
			</remarks>
		</summary>		
	</docu>	
~*)
    inStepID : INT;
    (*~
	<docu>
		<summary>
			If this value is false, step body is not executed and execution is moved to the next enabled step.
		</summary>				
	</docu>	
~*)
    inEnabled : BOOL;
    (*~
	<docu>
		<summary>
			Step description text.
		</summary>				
	</docu>	
~*)
    inStepDescription : STRING(254);
END_VAR
IF _suspenStepExecution THEN
	RETURN;
END_IF; 

Step := i_Step(inStepID := inStepID, inEnabled := inEnabled, inStepDescription := inStepDescription);
END_METHOD

(*~
	<docu>
		<summary>
			Completes the actually running step, when the `inCondition` parameter is `TRUE`.
			Method is typically called inside a step as the transition method.
		</summary>			
	</docu>	
~*)
METHOD PROTECTED FINAL StepCompleteWhen
VAR_INPUT
    (*~
	<docu>
		<summary>
			The condition under which the step is completed.
		</summary>			
	</docu>	
~*)
    inCondition : BOOL;
END_VAR
i_StepCompleteWhen(inCondition := inCondition);
END_METHOD

(*~
	<docu>
		<summary>
			This method s used to stop the clean cycle time measurement . 
				Method is typically called at the end of the sequence(e.g.in automat sequence )  .
		</summary>		
		<returns></returns>	
	</docu>	
~*)

METHOD PUBLIC StopCleanCycleTime
VAR_INPUT
END_VAR

VAR
	cleanCycleTime: TIME;
END_VAR
_stopCleanCycleTime:=_SequenceElapsedTime;

cleanCycleTime:=T#0S;
IF _stopCleanCycleTime>_startCleanCycleTime THEN
	cleanCycleTime:=_stopCleanCycleTime-_startCleanCycleTime;
 END_IF;

IF _cycleTimeAnalitics.FilterConstant = 0 THEN;
	_cycleTimeAnalitics.FilterConstant:=10;
END_IF;


IF _cycleTimeAnalitics.AverageCleanCycle = T#0S THEN
	_cycleTimeAnalitics.AverageCleanCycle:=_stopCleanCycleTime;
END_IF
_cycleTimeAnalitics.AverageCleanCycle:= (((_cycleTimeAnalitics.FilterConstant-1)*_cycleTimeAnalitics.AverageCleanCycle)+cleanCycleTime)/_cycleTimeAnalitics.FilterConstant;
END_METHOD

PROPERTY PUBLIC SuspendStepExecution : REFERENCE TO BOOL
GET
SuspendStepExecution ref=_suspenStepExecution;
END_GET
END_PROPERTY

PROPERTY Task : REFERENCE TO TcoTask
GET
Task REF= _task;
END_GET
END_PROPERTY

METHOD PUBLIC FINAL Timer_1 : BOOL
VAR_INPUT
	Condition : BOOL;
	PT : TIME;
END_VAR
_timer_1(IN:= Condition  and  not IsFreshState, PT:=PT);
Timer_1 := _timer_1.Q;
END_METHOD

METHOD PUBLIC FINAL Timer_2 : BOOL
VAR_INPUT
	Condition : BOOL;
	PT : TIME;
END_VAR
_timer_2(IN:= Condition and not IsFreshState, PT:=PT);
Timer_2 := _timer_2.Q;
END_METHOD

END_FUNCTION_BLOCK

// ---- Technology/CU00x/Automat/CU00xAutomatParalell_1_Task.TcPOU
FUNCTION_BLOCK CU00xAutomatParalell_1_Task EXTENDS TcoTaskedSequencer 

VAR
	_customTimer: TON;
END_VAR

Run();

(*~
	<docu>
		<summary>
			Main method of the sequener. Custom code needs to be placed here. The sequencer is executed by call of **Instance.Run()** method.
			This method is abstract, and it must be overridden in derived block.
		</summary>
	</docu>
~*)
METHOD PROTECTED Main : BOOL
// Takes mode (step/continous) from the parent controller
THIS^.ModeController.Mode := ParentSequence.ModeController.Mode;

IF (Step(1000, TRUE, 'PARALELL STEP - EXAMPLE OF TIMERS')) THEN
    //-------------------------------------    
		StepCompleteWhen(CurrentStep.Duration >= T#300mS);	
    //-------------------------------------
END_IF
IF (Step(1100, TRUE, 'PARALELL STEP - EXAMPLE OF TIMERS')) THEN
    //-------------------------------------    
		StepCompleteWhen(inCondition:=Timer_1(TRUE,T#100MS));	
    //-------------------------------------
END_IF
IF (Step(1200, TRUE, 'PARALELL STEP - EXAMPLE OF TIMERS')) THEN
    //-------------------------------------    
		StepCompleteWhen(inCondition:=Timer_1(TRUE,T#200MS));	
    //-------------------------------------
END_IF

IF THIS^.IsFreshState THEN
	_customTimer(IN:=FALSE);
END_IF
IF (Step(1300, TRUE, 'PARALELL STEP - EXAMPLE OF TIMERS')) THEN
    //-------------------------------------    

		_customTimer(IN:=TRUE,PT:=T#200MS);
		StepCompleteWhen(inCondition:=_customTimer.Q);	
    //-------------------------------------
END_IF


IF (Step(10000, TRUE, 'PARALELL TASK DONE')) THEN
    //-------------------------------------
    _task.DoneWhen(TRUE );
    //-------------------------------------	
END_IF
END_METHOD

PROPERTY ParentSequence : REFERENCE TO CU00xAutomatTask
GET
VAR
    _parentSequence : POINTER TO CU00xAutomatTask;
END_VAR
IF __QUERYPOINTER(Parent, _parentSequence) THEN 
    ParentSequence REF= _parentSequence^;              
END_IF
END_GET
END_PROPERTY

END_FUNCTION_BLOCK

// ---- Technology/CU00x/Data/CU00xDialogContent.TcPOU
FUNCTION_BLOCK CU00xDialogContent EXTENDS TcoCore.TcoInputDialogContentContainer
VAR_INPUT
END_VAR
VAR_OUTPUT
END_VAR
VAR
	{attribute addProperty Name "<#Recipe#>"}
	Recipe:STRING;
	{attribute addProperty Name "<#Qantity#>"}
	RequiredQuantity:INT;
	{attribute addProperty Name "<#Timeout#>"}
	Timeout:DATE_AND_TIME;
	{attribute addProperty Name "<#Exclude#>"}
	Exclude:BOOL;

END_VAR

END_FUNCTION_BLOCK

// ---- Technology/CU00x/Safety/Suspend/CU00xSuspendTask.TcPOU
FUNCTION_BLOCK CU00xSuspendTask EXTENDS CUBaseSuspend IMPLEMENTS ICUTask
VAR
	_sb : TcoCore.StringBuilder;
END_VAR

Run();

(*~
	<docu>
		<summary>
			Main method of the sequener. Custom code needs to be placed here. The sequencer is executed by call of **Instance.Run()** method.
			This method is abstract, and it must be overridden in derived block.
		</summary>
	</docu>
~*)
METHOD PROTECTED Main : BOOL
(*

	SUSPEND PROCESS 
	Following steps provide suspend actions for this controlled unit.
	Add components add write customized sequence according to your need.
*)

		
//
IF (Step(100, TRUE, '<#WAITING FOR START#>')) THEN
    //-------------------------------------    

    StepCompleteWhen(TRUE);
    //-------------------------------------
END_IF

